LIN {X 0,Y 577.255,Z 419.298,A -85,B 0,C 180,E1 20726.656,E2 20726.656} C_VEL
LIN {X 0,Y 577.259,Z 419.322,A -85,B 0,C 180,E1 20723.262,E2 20723.262} C_VEL
LIN {X 0,Y 577.272,Z 419.276,A -85,B 0,C 180,E1 20720.374,E2 20720.374} C_VEL
LIN {X 0,Y 577.266,Z 419.321,A -85,B 0,C 180,E1 20717.021,E2 20717.021} C_VEL
LIN {X 0,Y 577.313,Z 419.275,A -85,B 0,C 180,E1 20713.931,E2 20713.931} C_VEL
LIN {X 0,Y 577.267,Z 419.299,A -85,B 0,C 180,E1 20710.681,E2 20710.681} C_VEL
LIN {X 0,Y 577.322,Z 419.289,A -85,B 0,C 180,E1 20707.464,E2 20707.464} C_VEL
LIN {X 0,Y 577.275,Z 419.285,A -85,B 0,C 180,E1 20704.271,E2 20704.271} C_VEL
LIN {X 0,Y 577.307,Z 419.309,A -85,B 0,C 180,E1 20700.893,E2 20700.893} C_VEL
LIN {X 0,Y 577.308,Z 419.27,A -85,B 0,C 180,E1 20697.618,E2 20697.618} C_VEL
LIN {X 0,Y 577.29,Z 419.318,A -85,B 0,C 180,E1 20694.334,E2 20694.334} C_VEL
LIN {X 0,Y 577.307,Z 419.266,A -85,B 0,C 180,E1 20691.133,E2 20691.133} C_VEL
LIN {X 0,Y 577.298,Z 419.321,A -85,B 0,C 180,E1 20687.903,E2 20687.903} C_VEL
LIN {X 0,Y 577.31,Z 419.27,A -85,B 0,C 180,E1 20684.633,E2 20684.633} C_VEL
LIN {X 0,Y 577.313,Z 419.303,A -85,B 0,C 180,E1 20681.312,E2 20681.312} C_VEL
LIN {X 0,Y 577.312,Z 419.296,A -85,B 0,C 180,E1 20678.031,E2 20678.031} C_VEL
LIN {X 0,Y 577.295,Z 419.275,A -85,B 0,C 180,E1 20674.781,E2 20674.781} C_VEL
LIN {X 0,Y 577.312,Z 419.307,A -85,B 0,C 180,E1 20671.556,E2 20671.556} C_VEL
LIN {X 0,Y 577.315,Z 419.337,A -85,B 0,C 180,E1 20669.536,E2 20669.536} C_VEL
LIN {X 0,Y 578.617,Z 422.754,A -85,B 0,C 180,E1 20669.207,E2 20669.207} C_VEL
LIN {X 0,Y 581.308,Z 425.275,A -85,B 0,C 180,E1 20668.704,E2 20668.704} C_VEL
LIN {X 0,Y 582.264,Z 426.059,A -85,B 0,C 180,E1 20668.53,E2 20668.53} C_VEL
LIN {X 0,Y 584.624,Z 429.805,A -85,B 0,C 180,E1 20668.068,E2 20668.068} C_VEL
LIN {X 0,Y 587.281,Z 432.33,A -85,B 0,C 180,E1 20667.596,E2 20667.596} C_VEL
LIN {X 0,Y 590.354,Z 436.457,A -85,B 0,C 180,E1 20667.036,E2 20667.036} C_VEL
LIN {X 0,Y 592.909,Z 439.484,A -85,B 0,C 180,E1 20666.591,E2 20666.591} C_VEL
LIN {X 0,Y 603.214,Z 452.791,A -85,B 0,C 180,E1 20664.858,E2 20664.858} C_VEL
LIN {X 0,Y 615.76,Z 470.076,A -85,B 0,C 180,E1 20662.897,E2 20662.897} C_VEL
LIN {X 0,Y 629.647,Z 490.433,A -85,B 0,C 180,E1 20660.888,E2 20660.888} C_VEL
LIN {X 0,Y 623.894,Z 691.807,A -85,B 0,C 180,E1 20658.019,E2 20658.019} C_VEL
LIN {X 0,Y 623.038,Z 722.937,A -85,B 0,C 180,E1 20657.582,E2 20657.582} C_VEL
LIN {X 0,Y 622.123,Z 730.643,A -85,B 0,C 180,E1 20657.545,E2 20657.545} C_VEL
LIN {X 0,Y 617.355,Z 751.291,A -85,B 0,C 180,E1 20657.682,E2 20657.682} C_VEL
LIN {X 0,Y 616.661,Z 757.897,A -85,B 0,C 180,E1 20657.641,E2 20657.641} C_VEL
LIN {X 0,Y 612.677,Z 894.526,A -85,B 0,C 180,E1 20655.715,E2 20655.715} C_VEL
LIN {X 0,Y 611.264,Z 919.339,A -85,B 0,C 180,E1 20655.259,E2 20655.259} C_VEL
LIN {X 0,Y 609.02,Z 947.274,A -85,B 0,C 180,E1 20654.559,E2 20654.559} C_VEL
LIN {X 0,Y 606.96,Z 968.773,A -85,B 0,C 180,E1 20653.88,E2 20653.88} C_VEL
LIN {X 0,Y 604.761,Z 988.806,A -85,B 0,C 180,E1 20653.132,E2 20653.132} C_VEL
LIN {X 0,Y 602.479,Z 1008.004,A -85,B 0,C 180,E1 20652.299,E2 20652.299} C_VEL
LIN {X 0,Y 599.973,Z 1027.016,A -85,B 0,C 180,E1 20651.361,E2 20651.361} C_VEL
LIN {X 0,Y 597.085,Z 1047.482,A -85,B 0,C 180,E1 20650.215,E2 20650.215} C_VEL
LIN {X 0,Y 593.295,Z 1072.796,A -85,B 0,C 180,E1 20648.578,E2 20648.578} C_VEL
LIN {X 0,Y 590.157,Z 1092.691,A -85,B 0,C 180,E1 20647.098,E2 20647.098} C_VEL
LIN {X 0,Y 587.384,Z 1109.948,A -85,B 0,C 180,E1 20645.665,E2 20645.665} C_VEL
LIN {X 0,Y 584.673,Z 1126.712,A -85,B 0,C 180,E1 20644.122,E2 20644.122} C_VEL
LIN {X 0,Y 581.533,Z 1146.472,A -85,B 0,C 180,E1 20642.095,E2 20642.095} C_VEL
LIN {X 0,Y 578.659,Z 1164.633,A -85,B 0,C 180,E1 20639.96,E2 20639.96} C_VEL
LIN {X 0,Y 576.427,Z 1179.555,A -85,B 0,C 180,E1 20638.002,E2 20638.002} C_VEL
LIN {X 0,Y 574.396,Z 1193.881,A -85,B 0,C 180,E1 20635.91,E2 20635.91} C_VEL
LIN {X 0,Y 572.334,Z 1210.036,A -85,B 0,C 180,E1 20633.227,E2 20633.227} C_VEL
LIN {X 0,Y 570.945,Z 1222.042,A -85,B 0,C 180,E1 20630.934,E2 20630.934} C_VEL
LIN {X 0,Y 569.91,Z 1232.241,A -85,B 0,C 180,E1 20628.73,E2 20628.73} C_VEL
LIN {X 0,Y 569.079,Z 1242.76,A -85,B 0,C 180,E1 20626.12,E2 20626.12} C_VEL
LIN {X 0,Y 568.482,Z 1251.696,A -85,B 0,C 180,E1 20623.427,E2 20623.427} C_VEL
LIN {X 0,Y 568.187,Z 1257.937,A -85,B 0,C 180,E1 20621.164,E2 20621.164} C_VEL
LIN {X 0,Y 568.01,Z 1263.03,A -85,B 0,C 180,E1 20618.914,E2 20618.914} C_VEL
LIN {X 0,Y 567.949,Z 1267.415,A -85,B 0,C 180,E1 20616.371,E2 20616.371} C_VEL
LIN {X 0,Y 567.913,Z 1270.438,A -85,B 0,C 180,E1 20613.637,E2 20613.637} C_VEL
LIN {X 0,Y 567.901,Z 1271.703,A -85,B 0,C 180,E1 20611.314,E2 20611.314} C_VEL
LIN {X 0,Y 567.864,Z 1271.838,A -85,B 0,C 180,E1 20609.196,E2 20609.196} C_VEL
LIN {X 0,Y 567.911,Z 1270.98,A -85,B 0,C 180,E1 20607.076,E2 20607.076} C_VEL
LIN {X 0,Y 567.922,Z 1269.047,A -85,B 0,C 180,E1 20604.852,E2 20604.852} C_VEL
LIN {X 0,Y 567.957,Z 1265.815,A -85,B 0,C 180,E1 20602.518,E2 20602.518} C_VEL
LIN {X 0,Y 568.093,Z 1260.701,A -85,B 0,C 180,E1 20599.866,E2 20599.866} C_VEL
LIN {X 0,Y 568.382,Z 1253.797,A -85,B 0,C 180,E1 20597.197,E2 20597.197} C_VEL
LIN {X 0,Y 568.805,Z 1246.674,A -85,B 0,C 180,E1 20594.924,E2 20594.924} C_VEL
LIN {X 0,Y 569.368,Z 1238.677,A -85,B 0,C 180,E1 20592.739,E2 20592.739} C_VEL
LIN {X 0,Y 570.319,Z 1228.371,A -85,B 0,C 180,E1 20590.302,E2 20590.302} C_VEL
LIN {X 0,Y 571.731,Z 1214.972,A -85,B 0,C 180,E1 20587.593,E2 20587.593} C_VEL
LIN {X 0,Y 573.255,Z 1202.375,A -85,B 0,C 180,E1 20585.367,E2 20585.367} C_VEL
LIN {X 0,Y 575.105,Z 1188.883,A -85,B 0,C 180,E1 20583.242,E2 20583.242} C_VEL
LIN {X 0,Y 577.784,Z 1170.42,A -85,B 0,C 180,E1 20580.681,E2 20580.681} C_VEL
LIN {X 0,Y 580.26,Z 1154.409,A -85,B 0,C 180,E1 20578.727,E2 20578.727} C_VEL
LIN {X 0,Y 582.66,Z 1139.203,A -85,B 0,C 180,E1 20577.049,E2 20577.049} C_VEL
LIN {X 0,Y 585.444,Z 1122.069,A -85,B 0,C 180,E1 20575.343,E2 20575.343} C_VEL
LIN {X 0,Y 589.014,Z 1099.841,A -85,B 0,C 180,E1 20573.378,E2 20573.378} C_VEL
LIN {X 0,Y 592.274,Z 1079.106,A -85,B 0,C 180,E1 20571.782,E2 20571.782} C_VEL
LIN {X 0,Y 595.098,Z 1060.635,A -85,B 0,C 180,E1 20570.515,E2 20570.515} C_VEL
LIN {X 0,Y 598.159,Z 1039.88,A -85,B 0,C 180,E1 20569.249,E2 20569.249} C_VEL
LIN {X 0,Y 601.84,Z 1013.091,A -85,B 0,C 180,E1 20567.846,E2 20567.846} C_VEL
LIN {X 0,Y 604.399,Z 992.012,A -85,B 0,C 180,E1 20566.908,E2 20566.908} C_VEL
LIN {X 0,Y 606.726,Z 970.971,A -85,B 0,C 180,E1 20566.107,E2 20566.107} C_VEL
LIN {X 0,Y 608.75,Z 950.092,A -85,B 0,C 180,E1 20565.433,E2 20565.433} C_VEL
LIN {X 0,Y 610.629,Z 927.736,A -85,B 0,C 180,E1 20564.843,E2 20564.843} C_VEL
LIN {X 0,Y 612.456,Z 899.611,A -85,B 0,C 180,E1 20564.274,E2 20564.274} C_VEL
LIN {X 0,Y 614.038,Z 851.534,A -85,B 0,C 180,E1 20563.579,E2 20563.579} C_VEL
LIN {X 0,Y 620.348,Z 631.132,A -85,B 0,C 180,E1 20560.474,E2 20560.474} C_VEL
LIN {X 0,Y 624.432,Z 494.419,A -85,B 0,C 180,E1 20558.499,E2 20558.499} C_VEL
LIN {X 0,Y 611.394,Z 475.211,A -85,B 0,C 180,E1 20556.563,E2 20556.563} C_VEL
LIN {X 0,Y 598.761,Z 457.785,A -85,B 0,C 180,E1 20554.537,E2 20554.537} C_VEL
LIN {X 0,Y 588.143,Z 444.02,A -85,B 0,C 180,E1 20552.697,E2 20552.697} C_VEL
LIN {X 0,Y 584.586,Z 439.654,A -85,B 0,C 180,E1 20552.05,E2 20552.05} C_VEL
LIN {X 0,Y 583.05,Z 437.933,A -85,B 0,C 180,E1 20551.768,E2 20551.768} C_VEL
LIN {X 0,Y 579.933,Z 434.1,A -85,B 0,C 180,E1 20551.177,E2 20551.177} C_VEL
LIN {X 0,Y 578.924,Z 432.665,A -85,B 0,C 180,E1 20550.977,E2 20550.977} C_VEL
LIN {X 0,Y 575.807,Z 429.629,A -85,B 0,C 180,E1 20550.382,E2 20550.382} C_VEL
LIN {X 0,Y 573.999,Z 426.555,A -85,B 0,C 180,E1 20549.997,E2 20549.997} C_VEL
LIN {X 0,Y 571.024,Z 424.302,A -85,B 0,C 180,E1 20549.418,E2 20549.418} C_VEL
LIN {X 0,Y 569.558,Z 421.482,A -85,B 0,C 180,E1 20549.083,E2 20549.083} C_VEL
LIN {X 0,Y 569.316,Z 420.278,A -85,B 0,C 180,E1 20548.996,E2 20548.996} C_VEL
LIN {X 0,Y 569.359,Z 420.26,A -85,B 0,C 180,E1 20545.819,E2 20545.819} C_VEL
LIN {X 0,Y 569.316,Z 420.316,A -85,B 0,C 180,E1 20542.73,E2 20542.73} C_VEL
LIN {X 0,Y 569.344,Z 420.268,A -85,B 0,C 180,E1 20539.44,E2 20539.44} C_VEL
LIN {X 0,Y 569.315,Z 420.29,A -85,B 0,C 180,E1 20536.425,E2 20536.425} C_VEL
LIN {X 0,Y 569.329,Z 420.286,A -85,B 0,C 180,E1 20533.095,E2 20533.095} C_VEL
LIN {X 0,Y 569.315,Z 420.275,A -85,B 0,C 180,E1 20530.115,E2 20530.115} C_VEL
LIN {X 0,Y 569.318,Z 420.302,A -85,B 0,C 180,E1 20526.758,E2 20526.758} C_VEL
LIN {X 0,Y 569.317,Z 420.269,A -85,B 0,C 180,E1 20523.827,E2 20523.827} C_VEL
LIN {X 0,Y 569.314,Z 420.308,A -85,B 0,C 180,E1 20520.503,E2 20520.503} C_VEL
LIN {X 0,Y 569.316,Z 420.267,A -85,B 0,C 180,E1 20517.584,E2 20517.584} C_VEL
LIN {X 0,Y 569.312,Z 420.313,A -85,B 0,C 180,E1 20514.254,E2 20514.254} C_VEL
LIN {X 0,Y 569.312,Z 420.266,A -85,B 0,C 180,E1 20511.38,E2 20511.38} C_VEL
LIN {X 0,Y 569.306,Z 420.314,A -85,B 0,C 180,E1 20508.008,E2 20508.008} C_VEL
LIN {X 0,Y 569.31,Z 420.262,A -85,B 0,C 180,E1 20505.142,E2 20505.142} C_VEL
LIN {X 0,Y 569.303,Z 420.311,A -85,B 0,C 180,E1 20501.782,E2 20501.782} C_VEL
LIN {X 0,Y 569.319,Z 420.264,A -85,B 0,C 180,E1 20498.789,E2 20498.789} C_VEL
LIN {X 0,Y 569.295,Z 420.28,A -85,B 0,C 180,E1 20495.512,E2 20495.512} C_VEL
LIN {X 0,Y 569.333,Z 420.306,A -85,B 0,C 180,E1 20492.475,E2 20492.475} C_VEL
LIN {X 0,Y 569.34,Z 420.481,A -85,B 0,C 180,E1 20491.662,E2 20491.662} C_VEL
LIN {X 0,Y 570.676,Z 423.891,A -85,B 0,C 180,E1 20490.965,E2 20490.965} C_VEL
LIN {X 0,Y 572.177,Z 425.93,A -85,B 0,C 180,E1 20490.446,E2 20490.446} C_VEL
LIN {X 0,Y 575.339,Z 430.215,A -85,B 0,C 180,E1 20489.793,E2 20489.793} C_VEL
LIN {X 0,Y 577.584,Z 432.958,A -85,B 0,C 180,E1 20489.348,E2 20489.348} C_VEL
LIN {X 0,Y 585.42,Z 442.842,A -85,B 0,C 180,E1 20487.857,E2 20487.857} C_VEL
LIN {X 0,Y 590.299,Z 449.247,A -85,B 0,C 180,E1 20486.972,E2 20486.972} C_VEL
LIN {X 0,Y 600.49,Z 462.84,A -85,B 0,C 180,E1 20485.228,E2 20485.228} C_VEL
LIN {X 0,Y 612.268,Z 479.558,A -85,B 0,C 180,E1 20483.352,E2 20483.352} C_VEL
LIN {X 0,Y 624.192,Z 497.277,A -85,B 0,C 180,E1 20481.586,E2 20481.586} C_VEL
LIN {X 0,Y 624.554,Z 498.373,A -85,B 0,C 180,E1 20481.524,E2 20481.524} C_VEL
LIN {X 0,Y 618.433,Z 702.963,A -85,B 0,C 180,E1 20478.594,E2 20478.594} C_VEL
LIN {X 0,Y 612.66,Z 903.345,A -85,B 0,C 180,E1 20475.772,E2 20475.772} C_VEL
LIN {X 0,Y 611.318,Z 926.912,A -85,B 0,C 180,E1 20475.346,E2 20475.346} C_VEL
LIN {X 0,Y 609.063,Z 955.797,A -85,B 0,C 180,E1 20474.637,E2 20474.637} C_VEL
LIN {X 0,Y 606.994,Z 977.545,A -85,B 0,C 180,E1 20473.957,E2 20473.957} C_VEL
LIN {X 0,Y 604.718,Z 998.44,A -85,B 0,C 180,E1 20473.182,E2 20473.182} C_VEL
LIN {X 0,Y 602.468,Z 1017.534,A -85,B 0,C 180,E1 20472.356,E2 20472.356} C_VEL
LIN {X 0,Y 599.952,Z 1036.808,A -85,B 0,C 180,E1 20471.411,E2 20471.411} C_VEL
LIN {X 0,Y 597.09,Z 1057.377,A -85,B 0,C 180,E1 20470.265,E2 20470.265} C_VEL
LIN {X 0,Y 593.319,Z 1082.691,A -85,B 0,C 180,E1 20468.631,E2 20468.631} C_VEL
LIN {X 0,Y 590.173,Z 1102.602,A -85,B 0,C 180,E1 20467.151,E2 20467.151} C_VEL
LIN {X 0,Y 587.38,Z 1119.973,A -85,B 0,C 180,E1 20465.709,E2 20465.709} C_VEL
LIN {X 0,Y 584.596,Z 1137.198,A -85,B 0,C 180,E1 20464.12,E2 20464.12} C_VEL
LIN {X 0,Y 581.466,Z 1156.906,A -85,B 0,C 180,E1 20462.092,E2 20462.092} C_VEL
LIN {X 0,Y 578.6,Z 1175.014,A -85,B 0,C 180,E1 20459.957,E2 20459.957} C_VEL
LIN {X 0,Y 576.36,Z 1189.974,A -85,B 0,C 180,E1 20457.989,E2 20457.989} C_VEL
LIN {X 0,Y 574.263,Z 1204.905,A -85,B 0,C 180,E1 20455.799,E2 20455.799} C_VEL
LIN {X 0,Y 572.246,Z 1220.722,A -85,B 0,C 180,E1 20453.146,E2 20453.146} C_VEL
LIN {X 0,Y 570.918,Z 1232.282,A -85,B 0,C 180,E1 20450.929,E2 20450.929} C_VEL
LIN {X 0,Y 569.931,Z 1242,A -85,B 0,C 180,E1 20448.829,E2 20448.829} C_VEL
LIN {X 0,Y 569.148,Z 1251.779,A -85,B 0,C 180,E1 20446.417,E2 20446.417} C_VEL
LIN {X 0,Y 568.498,Z 1261.236,A -85,B 0,C 180,E1 20443.628,E2 20443.628} C_VEL
LIN {X 0,Y 568.204,Z 1267.555,A -85,B 0,C 180,E1 20441.363,E2 20441.363} C_VEL
LIN {X 0,Y 568.006,Z 1272.72,A -85,B 0,C 180,E1 20439.112,E2 20439.112} C_VEL
LIN {X 0,Y 567.949,Z 1276.862,A -85,B 0,C 180,E1 20436.771,E2 20436.771} C_VEL
LIN {X 0,Y 567.919,Z 1280.098,A -85,B 0,C 180,E1 20434.136,E2 20434.136} C_VEL
LIN {X 0,Y 567.902,Z 1281.691,A -85,B 0,C 180,E1 20431.409,E2 20431.409} C_VEL
LIN {X 0,Y 567.864,Z 1281.849,A -85,B 0,C 180,E1 20429.291,E2 20429.291} C_VEL
LIN {X 0,Y 567.911,Z 1281.013,A -85,B 0,C 180,E1 20427.172,E2 20427.172} C_VEL
LIN {X 0,Y 567.921,Z 1279.102,A -85,B 0,C 180,E1 20424.947,E2 20424.947} C_VEL
LIN {X 0,Y 567.957,Z 1275.894,A -85,B 0,C 180,E1 20422.614,E2 20422.614} C_VEL
LIN {X 0,Y 568.085,Z 1270.812,A -85,B 0,C 180,E1 20419.962,E2 20419.962} C_VEL
LIN {X 0,Y 568.369,Z 1263.95,A -85,B 0,C 180,E1 20417.294,E2 20417.294} C_VEL
LIN {X 0,Y 568.792,Z 1256.852,A -85,B 0,C 180,E1 20415.022,E2 20415.022} C_VEL
LIN {X 0,Y 569.352,Z 1248.81,A -85,B 0,C 180,E1 20412.818,E2 20412.818} C_VEL
LIN {X 0,Y 570.279,Z 1238.756,A -85,B 0,C 180,E1 20410.432,E2 20410.432} C_VEL
LIN {X 0,Y 571.697,Z 1225.279,A -85,B 0,C 180,E1 20407.693,E2 20407.693} C_VEL
LIN {X 0,Y 573.209,Z 1212.716,A -85,B 0,C 180,E1 20405.469,E2 20405.469} C_VEL
LIN {X 0,Y 575.051,Z 1199.261,A -85,B 0,C 180,E1 20403.344,E2 20403.344} C_VEL
LIN {X 0,Y 577.59,Z 1181.727,A -85,B 0,C 180,E1 20400.891,E2 20400.891} C_VEL
LIN {X 0,Y 580.209,Z 1164.739,A -85,B 0,C 180,E1 20398.81,E2 20398.81} C_VEL
LIN {X 0,Y 582.65,Z 1149.263,A -85,B 0,C 180,E1 20397.1,E2 20397.1} C_VEL
LIN {X 0,Y 585.394,Z 1132.354,A -85,B 0,C 180,E1 20395.416,E2 20395.416} C_VEL
LIN {X 0,Y 588.911,Z 1110.53,A -85,B 0,C 180,E1 20393.479,E2 20393.479} C_VEL
LIN {X 0,Y 592.253,Z 1089.208,A -85,B 0,C 180,E1 20391.835,E2 20391.835} C_VEL
LIN {X 0,Y 595.075,Z 1070.76,A -85,B 0,C 180,E1 20390.568,E2 20390.568} C_VEL
LIN {X 0,Y 597.874,Z 1051.659,A -85,B 0,C 180,E1 20389.401,E2 20389.401} C_VEL
LIN {X 0,Y 601.073,Z 1028.507,A -85,B 0,C 180,E1 20388.158,E2 20388.158} C_VEL
LIN {X 0,Y 604.185,Z 1003.202,A -85,B 0,C 180,E1 20387.011,E2 20387.011} C_VEL
LIN {X 0,Y 606.568,Z 981.579,A -85,B 0,C 180,E1 20386.183,E2 20386.183} C_VEL
LIN {X 0,Y 608.634,Z 960.325,A -85,B 0,C 180,E1 20385.495,E2 20385.495} C_VEL
LIN {X 0,Y 610.45,Z 938.806,A -85,B 0,C 180,E1 20384.923,E2 20384.923} C_VEL
LIN {X 0,Y 612.158,Z 913.923,A -85,B 0,C 180,E1 20384.401,E2 20384.401} C_VEL
LIN {X 0,Y 613.575,Z 876.43,A -85,B 0,C 180,E1 20383.838,E2 20383.838} C_VEL
LIN {X 0,Y 619.924,Z 652.053,A -85,B 0,C 180,E1 20380.685,E2 20380.685} C_VEL
LIN {X 0,Y 624.525,Z 497.803,A -85,B 0,C 180,E1 20378.463,E2 20378.463} C_VEL
LIN {X 0,Y 612.514,Z 479.937,A -85,B 0,C 180,E1 20376.689,E2 20376.689} C_VEL
LIN {X 0,Y 601.717,Z 464.605,A -85,B 0,C 180,E1 20374.981,E2 20374.981} C_VEL
LIN {X 0,Y 595.232,Z 455.876,A -85,B 0,C 180,E1 20373.897,E2 20373.897} C_VEL
LIN {X 0,Y 587.981,Z 446.173,A -85,B 0,C 180,E1 20372.621,E2 20372.621} C_VEL
LIN {X 0,Y 579.919,Z 435.911,A -85,B 0,C 180,E1 20371.12,E2 20371.12} C_VEL
LIN {X 0,Y 575.515,Z 430.361,A -85,B 0,C 180,E1 20370.255,E2 20370.255} C_VEL
LIN {X 0,Y 572.223,Z 426.049,A -85,B 0,C 180,E1 20369.58,E2 20369.58} C_VEL
LIN {X 0,Y 571.22,Z 424.558,A -85,B 0,C 180,E1 20369.234,E2 20369.234} C_VEL
LIN {X 0,Y 569.558,Z 421.437,A -85,B 0,C 180,E1 20368.523,E2 20368.523} C_VEL
LIN {X 0,Y 569.355,Z 420.292,A -85,B 0,C 180,E1 20368.305,E2 20368.305} C_VEL
LIN {X 0,Y 569.307,Z 420.267,A -85,B 0,C 180,E1 20365.153,E2 20365.153} C_VEL
LIN {X 0,Y 569.386,Z 420.287,A -85,B 0,C 180,E1 20361.965,E2 20361.965} C_VEL
LIN {X 0,Y 569.317,Z 420.29,A -85,B 0,C 180,E1 20358.748,E2 20358.748} C_VEL
LIN {X 0,Y 569.378,Z 420.258,A -85,B 0,C 180,E1 20355.586,E2 20355.586} C_VEL
LIN {X 0,Y 569.335,Z 420.309,A -85,B 0,C 180,E1 20352.372,E2 20352.372} C_VEL
LIN {X 0,Y 569.342,Z 420.255,A -85,B 0,C 180,E1 20348.992,E2 20348.992} C_VEL
LIN {X 0,Y 569.37,Z 420.309,A -85,B 0,C 180,E1 20345.846,E2 20345.846} C_VEL
LIN {X 0,Y 569.336,Z 420.258,A -85,B 0,C 180,E1 20342.516,E2 20342.516} C_VEL
LIN {X 0,Y 569.38,Z 420.299,A -85,B 0,C 180,E1 20339.296,E2 20339.296} C_VEL
LIN {X 0,Y 569.35,Z 420.263,A -85,B 0,C 180,E1 20335.964,E2 20335.964} C_VEL
LIN {X 0,Y 569.372,Z 420.285,A -85,B 0,C 180,E1 20332.635,E2 20332.635} C_VEL
LIN {X 0,Y 569.372,Z 420.279,A -85,B 0,C 180,E1 20329.272,E2 20329.272} C_VEL
LIN {X 0,Y 569.356,Z 420.267,A -85,B 0,C 180,E1 20325.974,E2 20325.974} C_VEL
LIN {X 0,Y 569.37,Z 420.305,A -85,B 0,C 180,E1 20322.735,E2 20322.735} C_VEL
LIN {X 0,Y 569.373,Z 420.258,A -85,B 0,C 180,E1 20319.33,E2 20319.33} C_VEL
LIN {X 0,Y 569.375,Z 420.286,A -85,B 0,C 180,E1 20316.067,E2 20316.067} C_VEL
LIN {X 0,Y 569.36,Z 420.294,A -85,B 0,C 180,E1 20312.701,E2 20312.701} C_VEL
LIN {X 0,Y 569.379,Z 420.415,A -85,B 0,C 180,E1 20310.87,E2 20310.87} C_VEL
LIN {X 0,Y 570.427,Z 423.392,A -85,B 0,C 180,E1 20310.606,E2 20310.606} C_VEL
LIN {X 0,Y 572.868,Z 425.927,A -85,B 0,C 180,E1 20310.111,E2 20310.111} C_VEL
LIN {X 0,Y 574.435,Z 427.024,A -85,B 0,C 180,E1 20309.812,E2 20309.812} C_VEL
LIN {X 0,Y 576.752,Z 430.772,A -85,B 0,C 180,E1 20309.327,E2 20309.327} C_VEL
LIN {X 0,Y 579.551,Z 433.39,A -85,B 0,C 180,E1 20308.801,E2 20308.801} C_VEL
LIN {X 0,Y 582.512,Z 437.438,A -85,B 0,C 180,E1 20308.228,E2 20308.228} C_VEL
LIN {X 0,Y 584.579,Z 439.588,A -85,B 0,C 180,E1 20307.852,E2 20307.852} C_VEL
LIN {X 0,Y 588.094,Z 443.946,A -85,B 0,C 180,E1 20307.213,E2 20307.213} C_VEL
LIN {X 0,Y 597.347,Z 455.975,A -85,B 0,C 180,E1 20305.602,E2 20305.602} C_VEL
LIN {X 0,Y 609.156,Z 472.052,A -85,B 0,C 180,E1 20303.69,E2 20303.69} C_VEL
LIN {X 0,Y 620.362,Z 488.375,A -85,B 0,C 180,E1 20301.997,E2 20301.997} C_VEL
LIN {X 0,Y 624.49,Z 494.843,A -85,B 0,C 180,E1 20301.396,E2 20301.396} C_VEL
LIN {X 0,Y 618.135,Z 706.554,A -85,B 0,C 180,E1 20298.365,E2 20298.365} C_VEL
LIN {X 0,Y 616.661,Z 757.897,A -85,B 0,C 180,E1 20297.641,E2 20297.641} C_VEL
LIN {X 0,Y 615.763,Z 765.6,A -85,B 0,C 180,E1 20297.602,E2 20297.602} C_VEL
LIN {X 0,Y 610.953,Z 786.238,A -85,B 0,C 180,E1 20297.745,E2 20297.745} C_VEL
LIN {X 0,Y 610.243,Z 792.846,A -85,B 0,C 180,E1 20297.705,E2 20297.705} C_VEL
LIN {X 0,Y 607.082,Z 895.175,A -85,B 0,C 180,E1 20296.248,E2 20296.248} C_VEL
LIN {X 0,Y 605.476,Z 922.029,A -85,B 0,C 180,E1 20295.747,E2 20295.747} C_VEL
LIN {X 0,Y 603.194,Z 948.425,A -85,B 0,C 180,E1 20295.066,E2 20295.066} C_VEL
LIN {X 0,Y 601.07,Z 969.618,A -85,B 0,C 180,E1 20294.389,E2 20294.389} C_VEL
LIN {X 0,Y 598.702,Z 990.192,A -85,B 0,C 180,E1 20293.611,E2 20293.611} C_VEL
LIN {X 0,Y 596.112,Z 1010.852,A -85,B 0,C 180,E1 20292.698,E2 20292.698} C_VEL
LIN {X 0,Y 592.764,Z 1035.101,A -85,B 0,C 180,E1 20291.46,E2 20291.46} C_VEL
LIN {X 0,Y 589.089,Z 1058.632,A -85,B 0,C 180,E1 20290.039,E2 20290.039} C_VEL
LIN {X 0,Y 586.085,Z 1077.213,A -85,B 0,C 180,E1 20288.766,E2 20288.766} C_VEL
LIN {X 0,Y 583.082,Z 1095.367,A -85,B 0,C 180,E1 20287.378,E2 20287.378} C_VEL
LIN {X 0,Y 579.896,Z 1114.212,A -85,B 0,C 180,E1 20285.771,E2 20285.771} C_VEL
LIN {X 0,Y 576.121,Z 1136.346,A -85,B 0,C 180,E1 20283.619,E2 20283.619} C_VEL
LIN {X 0,Y 573.324,Z 1152.994,A -85,B 0,C 180,E1 20281.784,E2 20281.784} C_VEL
LIN {X 0,Y 570.852,Z 1168.016,A -85,B 0,C 180,E1 20279.949,E2 20279.949} C_VEL
LIN {X 0,Y 568.127,Z 1185.441,A -85,B 0,C 180,E1 20277.575,E2 20277.575} C_VEL
LIN {X 0,Y 565.828,Z 1201.189,A -85,B 0,C 180,E1 20275.096,E2 20275.096} C_VEL
LIN {X 0,Y 564.233,Z 1213.323,A -85,B 0,C 180,E1 20272.948,E2 20272.948} C_VEL
LIN {X 0,Y 562.838,Z 1225.244,A -85,B 0,C 180,E1 20270.573,E2 20270.573} C_VEL
LIN {X 0,Y 561.603,Z 1237.509,A -85,B 0,C 180,E1 20267.725,E2 20267.725} C_VEL
LIN {X 0,Y 560.906,Z 1246.241,A -85,B 0,C 180,E1 20265.332,E2 20265.332} C_VEL
LIN {X 0,Y 560.455,Z 1253.303,A -85,B 0,C 180,E1 20263.067,E2 20263.067} C_VEL
LIN {X 0,Y 560.157,Z 1259.718,A -85,B 0,C 180,E1 20260.597,E2 20260.597} C_VEL
LIN {X 0,Y 559.957,Z 1265.342,A -85,B 0,C 180,E1 20257.802,E2 20257.802} C_VEL
LIN {X 0,Y 559.926,Z 1268.822,A -85,B 0,C 180,E1 20255.331,E2 20255.331} C_VEL
LIN {X 0,Y 559.91,Z 1270.847,A -85,B 0,C 180,E1 20253.074,E2 20253.074} C_VEL
LIN {X 0,Y 559.881,Z 1271.771,A -85,B 0,C 180,E1 20251.026,E2 20251.026} C_VEL
LIN {X 0,Y 559.873,Z 1271.792,A -85,B 0,C 180,E1 20248.98,E2 20248.98} C_VEL
LIN {X 0,Y 559.911,Z 1270.911,A -85,B 0,C 180,E1 20246.932,E2 20246.932} C_VEL
LIN {X 0,Y 559.923,Z 1268.929,A -85,B 0,C 180,E1 20244.675,E2 20244.675} C_VEL
LIN {X 0,Y 559.96,Z 1265.491,A -85,B 0,C 180,E1 20242.204,E2 20242.204} C_VEL
LIN {X 0,Y 560.149,Z 1259.953,A -85,B 0,C 180,E1 20239.409,E2 20239.409} C_VEL
LIN {X 0,Y 560.448,Z 1253.492,A -85,B 0,C 180,E1 20236.908,E2 20236.908} C_VEL
LIN {X 0,Y 560.896,Z 1246.318,A -85,B 0,C 180,E1 20234.6,E2 20234.6} C_VEL
LIN {X 0,Y 561.573,Z 1237.862,A -85,B 0,C 180,E1 20232.278,E2 20232.278} C_VEL
LIN {X 0,Y 562.803,Z 1225.581,A -85,B 0,C 180,E1 20229.408,E2 20229.408} C_VEL
LIN {X 0,Y 564.168,Z 1213.82,A -85,B 0,C 180,E1 20227.055,E2 20227.055} C_VEL
LIN {X 0,Y 565.745,Z 1201.734,A -85,B 0,C 180,E1 20224.906,E2 20224.906} C_VEL
LIN {X 0,Y 567.92,Z 1186.761,A -85,B 0,C 180,E1 20222.535,E2 20222.535} C_VEL
LIN {X 0,Y 570.616,Z 1169.546,A -85,B 0,C 180,E1 20220.157,E2 20220.157} C_VEL
LIN {X 0,Y 573.088,Z 1154.433,A -85,B 0,C 180,E1 20218.294,E2 20218.294} C_VEL
LIN {X 0,Y 575.716,Z 1138.688,A -85,B 0,C 180,E1 20216.54,E2 20216.54} C_VEL
LIN {X 0,Y 578.848,Z 1120.395,A -85,B 0,C 180,E1 20214.709,E2 20214.709} C_VEL
LIN {X 0,Y 582.679,Z 1097.76,A -85,B 0,C 180,E1 20212.722,E2 20212.722} C_VEL
LIN {X 0,Y 585.811,Z 1078.871,A -85,B 0,C 180,E1 20211.264,E2 20211.264} C_VEL
LIN {X 0,Y 588.794,Z 1060.419,A -85,B 0,C 180,E1 20209.986,E2 20209.986} C_VEL
LIN {X 0,Y 591.945,Z 1040.055,A -85,B 0,C 180,E1 20208.736,E2 20208.736} C_VEL
LIN {X 0,Y 595.666,Z 1014.294,A -85,B 0,C 180,E1 20207.372,E2 20207.372} C_VEL
LIN {X 0,Y 598.557,Z 991.428,A -85,B 0,C 180,E1 20206.349,E2 20206.349} C_VEL
LIN {X 0,Y 600.915,Z 971.041,A -85,B 0,C 180,E1 20205.571,E2 20205.571} C_VEL
LIN {X 0,Y 603.032,Z 950.05,A -85,B 0,C 180,E1 20204.891,E2 20204.891} C_VEL
LIN {X 0,Y 604.996,Z 927.537,A -85,B 0,C 180,E1 20204.295,E2 20204.295} C_VEL
LIN {X 0,Y 606.923,Z 898.692,A -85,B 0,C 180,E1 20203.716,E2 20203.716} C_VEL
LIN {X 0,Y 608.642,Z 847.708,A -85,B 0,C 180,E1 20202.977,E2 20202.977} C_VEL
LIN {X 0,Y 615.268,Z 627.748,A -85,B 0,C 180,E1 20199.856,E2 20199.856} C_VEL
LIN {X 0,Y 619.331,Z 498.457,A -85,B 0,C 180,E1 20197.975,E2 20197.975} C_VEL
LIN {X 0,Y 606.402,Z 479.36,A -85,B 0,C 180,E1 20196.003,E2 20196.003} C_VEL
LIN {X 0,Y 592.009,Z 459.543,A -85,B 0,C 180,E1 20193.612,E2 20193.612} C_VEL
LIN {X 0,Y 585.035,Z 450.699,A -85,B 0,C 180,E1 20192.37,E2 20192.37} C_VEL
LIN {X 0,Y 580.351,Z 444.972,A -85,B 0,C 180,E1 20191.498,E2 20191.498} C_VEL
LIN {X 0,Y 576.818,Z 440.49,A -85,B 0,C 180,E1 20190.813,E2 20190.813} C_VEL
LIN {X 0,Y 572.742,Z 436.034,A -85,B 0,C 180,E1 20190.011,E2 20190.011} C_VEL
LIN {X 0,Y 571.245,Z 433.754,A -85,B 0,C 180,E1 20189.693,E2 20189.693} C_VEL
LIN {X 0,Y 568.122,Z 430.903,A -85,B 0,C 180,E1 20189.062,E2 20189.062} C_VEL
LIN {X 0,Y 566.3,Z 427.687,A -85,B 0,C 180,E1 20188.645,E2 20188.645} C_VEL
LIN {X 0,Y 563.23,Z 425.419,A -85,B 0,C 180,E1 20188.006,E2 20188.006} C_VEL
LIN {X 0,Y 561.67,Z 422.586,A -85,B 0,C 180,E1 20187.628,E2 20187.628} C_VEL
LIN {X 0,Y 561.392,Z 421.296,A -85,B 0,C 180,E1 20187.515,E2 20187.515} C_VEL
LIN {X 0,Y 561.401,Z 421.258,A -85,B 0,C 180,E1 20184.407,E2 20184.407} C_VEL
LIN {X 0,Y 561.379,Z 421.26,A -85,B 0,C 180,E1 20181.197,E2 20181.197} C_VEL
LIN {X 0,Y 561.406,Z 421.291,A -85,B 0,C 180,E1 20178.161,E2 20178.161} C_VEL
LIN {X 0,Y 561.366,Z 421.247,A -85,B 0,C 180,E1 20174.862,E2 20174.862} C_VEL
LIN {X 0,Y 561.417,Z 421.301,A -85,B 0,C 180,E1 20171.819,E2 20171.819} C_VEL
LIN {X 0,Y 561.363,Z 421.247,A -85,B 0,C 180,E1 20168.605,E2 20168.605} C_VEL
LIN {X 0,Y 561.411,Z 421.3,A -85,B 0,C 180,E1 20165.622,E2 20165.622} C_VEL
LIN {X 0,Y 561.36,Z 421.249,A -85,B 0,C 180,E1 20162.348,E2 20162.348} C_VEL
LIN {X 0,Y 561.423,Z 421.294,A -85,B 0,C 180,E1 20159.286,E2 20159.286} C_VEL
LIN {X 0,Y 561.356,Z 421.253,A -85,B 0,C 180,E1 20156.017,E2 20156.017} C_VEL
LIN {X 0,Y 561.441,Z 421.284,A -85,B 0,C 180,E1 20152.839,E2 20152.839} C_VEL
LIN {X 0,Y 561.354,Z 421.26,A -85,B 0,C 180,E1 20149.636,E2 20149.636} C_VEL
LIN {X 0,Y 561.406,Z 421.269,A -85,B 0,C 180,E1 20146.403,E2 20146.403} C_VEL
LIN {X 0,Y 561.356,Z 421.272,A -85,B 0,C 180,E1 20143.373,E2 20143.373} C_VEL
LIN {X 0,Y 561.392,Z 421.249,A -85,B 0,C 180,E1 20140.112,E2 20140.112} C_VEL
LIN {X 0,Y 561.356,Z 421.303,A -85,B 0,C 180,E1 20137.151,E2 20137.151} C_VEL
LIN {X 0,Y 561.386,Z 421.255,A -85,B 0,C 180,E1 20133.842,E2 20133.842} C_VEL
LIN {X 0,Y 561.362,Z 421.364,A -85,B 0,C 180,E1 20133.059,E2 20133.059} C_VEL
LIN {X 0,Y 562.59,Z 424.593,A -85,B 0,C 180,E1 20132.362,E2 20132.362} C_VEL
LIN {X 0,Y 564.373,Z 426.58,A -85,B 0,C 180,E1 20131.854,E2 20131.854} C_VEL
LIN {X 0,Y 567.267,Z 430.737,A -85,B 0,C 180,E1 20131.207,E2 20131.207} C_VEL
LIN {X 0,Y 569.664,Z 433.205,A -85,B 0,C 180,E1 20130.71,E2 20130.71} C_VEL
LIN {X 0,Y 573.277,Z 437.799,A -85,B 0,C 180,E1 20129.962,E2 20129.962} C_VEL
LIN {X 0,Y 582.806,Z 450.095,A -85,B 0,C 180,E1 20128.101,E2 20128.101} C_VEL
LIN {X 0,Y 587.875,Z 456.785,A -85,B 0,C 180,E1 20127.17,E2 20127.17} C_VEL
LIN {X 0,Y 597.266,Z 469.415,A -85,B 0,C 180,E1 20125.538,E2 20125.538} C_VEL
LIN {X 0,Y 610.901,Z 488.879,A -85,B 0,C 180,E1 20123.344,E2 20123.344} C_VEL
LIN {X 0,Y 619.452,Z 502.2,A -85,B 0,C 180,E1 20122.05,E2 20122.05} C_VEL
LIN {X 0,Y 612.928,Z 710.012,A -85,B 0,C 180,E1 20119.056,E2 20119.056} C_VEL
LIN {X 0,Y 607.076,Z 903.364,A -85,B 0,C 180,E1 20116.313,E2 20116.313} C_VEL
LIN {X 0,Y 605.654,Z 927.281,A -85,B 0,C 180,E1 20115.879,E2 20115.879} C_VEL
LIN {X 0,Y 603.313,Z 955.925,A -85,B 0,C 180,E1 20115.17,E2 20115.17} C_VEL
LIN {X 0,Y 601.092,Z 978.171,A -85,B 0,C 180,E1 20114.469,E2 20114.469} C_VEL
LIN {X 0,Y 598.818,Z 998.119,A -85,B 0,C 180,E1 20113.725,E2 20113.725} C_VEL
LIN {X 0,Y 596.436,Z 1017.445,A -85,B 0,C 180,E1 20112.887,E2 20112.887} C_VEL
LIN {X 0,Y 593.811,Z 1036.588,A -85,B 0,C 180,E1 20111.944,E2 20111.944} C_VEL
LIN {X 0,Y 590.792,Z 1057.286,A -85,B 0,C 180,E1 20110.784,E2 20110.784} C_VEL
LIN {X 0,Y 586.87,Z 1082.596,A -85,B 0,C 180,E1 20109.142,E2 20109.142} C_VEL
LIN {X 0,Y 583.61,Z 1102.282,A -85,B 0,C 180,E1 20107.67,E2 20107.67} C_VEL
LIN {X 0,Y 580.743,Z 1119.26,A -85,B 0,C 180,E1 20106.252,E2 20106.252} C_VEL
LIN {X 0,Y 577.872,Z 1136.087,A -85,B 0,C 180,E1 20104.694,E2 20104.694} C_VEL
LIN {X 0,Y 574.954,Z 1153.291,A -85,B 0,C 180,E1 20102.924,E2 20102.924} C_VEL
LIN {X 0,Y 571.461,Z 1174.167,A -85,B 0,C 180,E1 20100.487,E2 20100.487} C_VEL
LIN {X 0,Y 569.141,Z 1188.863,A -85,B 0,C 180,E1 20098.541,E2 20098.541} C_VEL
LIN {X 0,Y 567.023,Z 1202.801,A -85,B 0,C 180,E1 20096.492,E2 20096.492} C_VEL
LIN {X 0,Y 564.886,Z 1218.401,A -85,B 0,C 180,E1 20093.908,E2 20093.908} C_VEL
LIN {X 0,Y 563.262,Z 1231.25,A -85,B 0,C 180,E1 20091.446,E2 20091.446} C_VEL
LIN {X 0,Y 562.196,Z 1241.081,A -85,B 0,C 180,E1 20089.314,E2 20089.314} C_VEL
LIN {X 0,Y 561.357,Z 1250.123,A -85,B 0,C 180,E1 20087.088,E2 20087.088} C_VEL
LIN {X 0,Y 560.697,Z 1258.993,A -85,B 0,C 180,E1 20084.559,E2 20084.559} C_VEL
LIN {X 0,Y 560.264,Z 1267.044,A -85,B 0,C 180,E1 20081.735,E2 20081.735} C_VEL
LIN {X 0,Y 560.02,Z 1272.304,A -85,B 0,C 180,E1 20079.451,E2 20079.451} C_VEL
LIN {X 0,Y 559.967,Z 1276.38,A -85,B 0,C 180,E1 20077.177,E2 20077.177} C_VEL
LIN {X 0,Y 559.919,Z 1279.448,A -85,B 0,C 180,E1 20074.811,E2 20074.811} C_VEL
LIN {X 0,Y 559.911,Z 1281.55,A -85,B 0,C 180,E1 20072.044,E2 20072.044} C_VEL
LIN {X 0,Y 559.865,Z 1281.871,A -85,B 0,C 180,E1 20069.383,E2 20069.383} C_VEL
LIN {X 0,Y 559.909,Z 1281.081,A -85,B 0,C 180,E1 20067.233,E2 20067.233} C_VEL
LIN {X 0,Y 559.921,Z 1279.213,A -85,B 0,C 180,E1 20064.977,E2 20064.977} C_VEL
LIN {X 0,Y 559.964,Z 1276.21,A -85,B 0,C 180,E1 20062.714,E2 20062.714} C_VEL
LIN {X 0,Y 560.051,Z 1271.672,A -85,B 0,C 180,E1 20060.232,E2 20060.232} C_VEL
LIN {X 0,Y 560.377,Z 1264.556,A -85,B 0,C 180,E1 20057.32,E2 20057.32} C_VEL
LIN {X 0,Y 560.864,Z 1256.852,A -85,B 0,C 180,E1 20054.805,E2 20054.805} C_VEL
LIN {X 0,Y 561.467,Z 1248.885,A -85,B 0,C 180,E1 20052.589,E2 20052.589} C_VEL
LIN {X 0,Y 562.466,Z 1238.758,A -85,B 0,C 180,E1 20050.149,E2 20050.149} C_VEL
LIN {X 0,Y 563.987,Z 1225.278,A -85,B 0,C 180,E1 20047.372,E2 20047.372} C_VEL
LIN {X 0,Y 565.606,Z 1212.714,A -85,B 0,C 180,E1 20045.117,E2 20045.117} C_VEL
LIN {X 0,Y 567.556,Z 1199.259,A -85,B 0,C 180,E1 20042.963,E2 20042.963} C_VEL
LIN {X 0,Y 570.365,Z 1181.123,A -85,B 0,C 180,E1 20040.404,E2 20040.404} C_VEL
LIN {X 0,Y 573.033,Z 1164.761,A -85,B 0,C 180,E1 20038.377,E2 20038.377} C_VEL
LIN {X 0,Y 575.569,Z 1149.569,A -85,B 0,C 180,E1 20036.679,E2 20036.679} C_VEL
LIN {X 0,Y 578.36,Z 1133.256,A -85,B 0,C 180,E1 20035.032,E2 20035.032} C_VEL
LIN {X 0,Y 581.912,Z 1112.493,A -85,B 0,C 180,E1 20033.152,E2 20033.152} C_VEL
LIN {X 0,Y 585.63,Z 1089.94,A -85,B 0,C 180,E1 20031.386,E2 20031.386} C_VEL
LIN {X 0,Y 588.573,Z 1071.512,A -85,B 0,C 180,E1 20030.109,E2 20030.109} C_VEL
LIN {X 0,Y 591.598,Z 1051.765,A -85,B 0,C 180,E1 20028.892,E2 20028.892} C_VEL
LIN {X 0,Y 594.829,Z 1029.426,A -85,B 0,C 180,E1 20027.682,E2 20027.682} C_VEL
LIN {X 0,Y 598.234,Z 1003.121,A -85,B 0,C 180,E1 20026.478,E2 20026.478} C_VEL
LIN {X 0,Y 600.73,Z 981.491,A -85,B 0,C 180,E1 20025.646,E2 20025.646} C_VEL
LIN {X 0,Y 602.862,Z 960.442,A -85,B 0,C 180,E1 20024.962,E2 20024.962} C_VEL
LIN {X 0,Y 604.75,Z 939.042,A -85,B 0,C 180,E1 20024.389,E2 20024.389} C_VEL
LIN {X 0,Y 606.474,Z 914.973,A -85,B 0,C 180,E1 20023.879,E2 20023.879} C_VEL
LIN {X 0,Y 607.97,Z 878.645,A -85,B 0,C 180,E1 20023.324,E2 20023.324} C_VEL
LIN {X 0,Y 614.641,Z 654.12,A -85,B 0,C 180,E1 20020.147,E2 20020.147} C_VEL
LIN {X 0,Y 619.41,Z 501.851,A -85,B 0,C 180,E1 20017.94,E2 20017.94} C_VEL
LIN {X 0,Y 606.991,Z 483.206,A -85,B 0,C 180,E1 20016.05,E2 20016.05} C_VEL
LIN {X 0,Y 593.948,Z 464.767,A -85,B 0,C 180,E1 20013.902,E2 20013.902} C_VEL
LIN {X 0,Y 584.636,Z 452.504,A -85,B 0,C 180,E1 20012.25,E2 20012.25} C_VEL
LIN {X 0,Y 577.014,Z 442.679,A -85,B 0,C 180,E1 20010.802,E2 20010.802} C_VEL
LIN {X 0,Y 572.543,Z 437.042,A -85,B 0,C 180,E1 20009.907,E2 20009.907} C_VEL
LIN {X 0,Y 568.638,Z 431.999,A -85,B 0,C 180,E1 20009.091,E2 20009.091} C_VEL
LIN {X 0,Y 565.309,Z 428.206,A -85,B 0,C 180,E1 20008.382,E2 20008.382} C_VEL
LIN {X 0,Y 563.876,Z 426.106,A -85,B 0,C 180,E1 20008.057,E2 20008.057} C_VEL
LIN {X 0,Y 561.693,Z 422.759,A -85,B 0,C 180,E1 20007.226,E2 20007.226} C_VEL
LIN {X 0,Y 561.367,Z 421.281,A -85,B 0,C 180,E1 20006.899,E2 20006.899} C_VEL
LIN {X 0,Y 561.41,Z 421.279,A -85,B 0,C 180,E1 20003.624,E2 20003.624} C_VEL
LIN {X 0,Y 561.376,Z 421.253,A -85,B 0,C 180,E1 20000.651,E2 20000.651} C_VEL
LIN {X 0,Y 561.407,Z 421.298,A -85,B 0,C 180,E1 19997.304,E2 19997.304} C_VEL
LIN {X 0,Y 561.4,Z 421.248,A -85,B 0,C 180,E1 19994.228,E2 19994.228} C_VEL
LIN {X 0,Y 561.395,Z 421.279,A -85,B 0,C 180,E1 19990.883,E2 19990.883} C_VEL
LIN {X 0,Y 561.441,Z 421.257,A -85,B 0,C 180,E1 19987.676,E2 19987.676} C_VEL
LIN {X 0,Y 561.395,Z 421.265,A -85,B 0,C 180,E1 19984.495,E2 19984.495} C_VEL
LIN {X 0,Y 561.442,Z 421.269,A -85,B 0,C 180,E1 19981.225,E2 19981.225} C_VEL
LIN {X 0,Y 561.411,Z 421.251,A -85,B 0,C 180,E1 19977.959,E2 19977.959} C_VEL
LIN {X 0,Y 561.419,Z 421.295,A -85,B 0,C 180,E1 19974.481,E2 19974.481} C_VEL
LIN {X 0,Y 561.431,Z 421.241,A -85,B 0,C 180,E1 19971.279,E2 19971.279} C_VEL
LIN {X 0,Y 561.42,Z 421.299,A -85,B 0,C 180,E1 19967.973,E2 19967.973} C_VEL
LIN {X 0,Y 561.429,Z 421.243,A -85,B 0,C 180,E1 19964.717,E2 19964.717} C_VEL
LIN {X 0,Y 561.435,Z 421.277,A -85,B 0,C 180,E1 19961.302,E2 19961.302} C_VEL
LIN {X 0,Y 561.43,Z 421.273,A -85,B 0,C 180,E1 19957.927,E2 19957.927} C_VEL
LIN {X 0,Y 561.418,Z 421.248,A -85,B 0,C 180,E1 19954.694,E2 19954.694} C_VEL
LIN {X 0,Y 561.448,Z 421.431,A -85,B 0,C 180,E1 19952.336,E2 19952.336} C_VEL
LIN {X 0,Y 562.422,Z 424.249,A -85,B 0,C 180,E1 19952.071,E2 19952.071} C_VEL
LIN {X 0,Y 564.756,Z 426.827,A -85,B 0,C 180,E1 19951.558,E2 19951.558} C_VEL
LIN {X 0,Y 566.594,Z 428.047,A -85,B 0,C 180,E1 19951.184,E2 19951.184} C_VEL
LIN {X 0,Y 568.707,Z 431.588,A -85,B 0,C 180,E1 19950.708,E2 19950.708} C_VEL
LIN {X 0,Y 571.838,Z 434.431,A -85,B 0,C 180,E1 19950.081,E2 19950.081} C_VEL
LIN {X 0,Y 574.792,Z 438.512,A -85,B 0,C 180,E1 19949.472,E2 19949.472} C_VEL
LIN {X 0,Y 576.868,Z 440.559,A -85,B 0,C 180,E1 19949.074,E2 19949.074} C_VEL
LIN {X 0,Y 580.29,Z 444.925,A -85,B 0,C 180,E1 19948.411,E2 19948.411} C_VEL
LIN {X 0,Y 582.156,Z 447.164,A -85,B 0,C 180,E1 19948.061,E2 19948.061} C_VEL
LIN {X 0,Y 587.485,Z 453.774,A -85,B 0,C 180,E1 19947.087,E2 19947.087} C_VEL
LIN {X 0,Y 596.638,Z 465.769,A -85,B 0,C 180,E1 19945.497,E2 19945.497} C_VEL
LIN {X 0,Y 609.74,Z 484.146,A -85,B 0,C 180,E1 19943.38,E2 19943.38} C_VEL
LIN {X 0,Y 619.387,Z 498.754,A -85,B 0,C 180,E1 19941.921,E2 19941.921} C_VEL
LIN {X 0,Y 612.652,Z 712.627,A -85,B 0,C 180,E1 19938.841,E2 19938.841} C_VEL
LIN {X 0,Y 610.243,Z 792.846,A -85,B 0,C 180,E1 19937.705,E2 19937.705} C_VEL
LIN {X 0,Y 609.334,Z 800.551,A -85,B 0,C 180,E1 19937.667,E2 19937.667} C_VEL
LIN {X 0,Y 604.513,Z 821.189,A -85,B 0,C 180,E1 19937.813,E2 19937.813} C_VEL
LIN {X 0,Y 603.808,Z 827.797,A -85,B 0,C 180,E1 19937.773,E2 19937.773} C_VEL
LIN {X 0,Y 601.512,Z 896.456,A -85,B 0,C 180,E1 19936.782,E2 19936.782} C_VEL
LIN {X 0,Y 599.663,Z 924.651,A -85,B 0,C 180,E1 19936.238,E2 19936.238} C_VEL
LIN {X 0,Y 597.461,Z 949.163,A -85,B 0,C 180,E1 19935.595,E2 19935.595} C_VEL
LIN {X 0,Y 595.311,Z 969.725,A -85,B 0,C 180,E1 19934.934,E2 19934.934} C_VEL
LIN {X 0,Y 592.843,Z 990.297,A -85,B 0,C 180,E1 19934.153,E2 19934.153} C_VEL
LIN {X 0,Y 590.135,Z 1011.004,A -85,B 0,C 180,E1 19933.233,E2 19933.233} C_VEL
LIN {X 0,Y 586.69,Z 1034.919,A -85,B 0,C 180,E1 19932.006,E2 19932.006} C_VEL
LIN {X 0,Y 582.809,Z 1058.732,A -85,B 0,C 180,E1 19930.56,E2 19930.56} C_VEL
LIN {X 0,Y 579.66,Z 1077.313,A -85,B 0,C 180,E1 19929.278,E2 19929.278} C_VEL
LIN {X 0,Y 576.615,Z 1094.735,A -85,B 0,C 180,E1 19927.933,E2 19927.933} C_VEL
LIN {X 0,Y 573.361,Z 1113.001,A -85,B 0,C 180,E1 19926.367,E2 19926.367} C_VEL
LIN {X 0,Y 569.463,Z 1134.683,A -85,B 0,C 180,E1 19924.266,E2 19924.266} C_VEL
LIN {X 0,Y 566.27,Z 1152.536,A -85,B 0,C 180,E1 19922.287,E2 19922.287} C_VEL
LIN {X 0,Y 563.664,Z 1167.494,A -85,B 0,C 180,E1 19920.444,E2 19920.444} C_VEL
LIN {X 0,Y 561.095,Z 1183.003,A -85,B 0,C 180,E1 19918.318,E2 19918.318} C_VEL
LIN {X 0,Y 558.462,Z 1199.921,A -85,B 0,C 180,E1 19915.678,E2 19915.678} C_VEL
LIN {X 0,Y 556.613,Z 1212.865,A -85,B 0,C 180,E1 19913.371,E2 19913.371} C_VEL
LIN {X 0,Y 555.171,Z 1224.17,A -85,B 0,C 180,E1 19911.101,E2 19911.101} C_VEL
LIN {X 0,Y 553.857,Z 1236.272,A -85,B 0,C 180,E1 19908.31,E2 19908.31} C_VEL
LIN {X 0,Y 553.018,Z 1245.643,A -85,B 0,C 180,E1 19905.739,E2 19905.739} C_VEL
LIN {X 0,Y 552.523,Z 1252.609,A -85,B 0,C 180,E1 19903.503,E2 19903.503} C_VEL
LIN {X 0,Y 552.216,Z 1258.448,A -85,B 0,C 180,E1 19901.28,E2 19901.28} C_VEL
LIN {X 0,Y 552.016,Z 1263.439,A -85,B 0,C 180,E1 19898.964,E2 19898.964} C_VEL
LIN {X 0,Y 551.945,Z 1267.995,A -85,B 0,C 180,E1 19896.138,E2 19896.138} C_VEL
LIN {X 0,Y 551.913,Z 1270.575,A -85,B 0,C 180,E1 19893.534,E2 19893.534} C_VEL
LIN {X 0,Y 551.897,Z 1271.725,A -85,B 0,C 180,E1 19891.249,E2 19891.249} C_VEL
LIN {X 0,Y 551.866,Z 1271.837,A -85,B 0,C 180,E1 19889.173,E2 19889.173} C_VEL
LIN {X 0,Y 551.911,Z 1270.978,A -85,B 0,C 180,E1 19886.991,E2 19886.991} C_VEL
LIN {X 0,Y 551.923,Z 1269.039,A -85,B 0,C 180,E1 19884.702,E2 19884.702} C_VEL
LIN {X 0,Y 551.958,Z 1265.807,A -85,B 0,C 180,E1 19882.3,E2 19882.3} C_VEL
LIN {X 0,Y 552.148,Z 1260.598,A -85,B 0,C 180,E1 19879.524,E2 19879.524} C_VEL
LIN {X 0,Y 552.475,Z 1253.792,A -85,B 0,C 180,E1 19876.822,E2 19876.822} C_VEL
LIN {X 0,Y 552.944,Z 1246.668,A -85,B 0,C 180,E1 19874.481,E2 19874.481} C_VEL
LIN {X 0,Y 553.624,Z 1238.669,A -85,B 0,C 180,E1 19872.232,E2 19872.232} C_VEL
LIN {X 0,Y 554.751,Z 1228.04,A -85,B 0,C 180,E1 19869.647,E2 19869.647} C_VEL
LIN {X 0,Y 556.334,Z 1214.961,A -85,B 0,C 180,E1 19866.937,E2 19866.937} C_VEL
LIN {X 0,Y 558.075,Z 1202.363,A -85,B 0,C 180,E1 19864.651,E2 19864.651} C_VEL
LIN {X 0,Y 560.242,Z 1188.169,A -85,B 0,C 180,E1 19862.357,E2 19862.357} C_VEL
LIN {X 0,Y 563.203,Z 1170.359,A -85,B 0,C 180,E1 19859.838,E2 19859.838} C_VEL
LIN {X 0,Y 565.905,Z 1154.674,A -85,B 0,C 180,E1 19857.876,E2 19857.876} C_VEL
LIN {X 0,Y 568.712,Z 1138.777,A -85,B 0,C 180,E1 19856.084,E2 19856.084} C_VEL
LIN {X 0,Y 571.919,Z 1120.942,A -85,B 0,C 180,E1 19854.278,E2 19854.278} C_VEL
LIN {X 0,Y 576.079,Z 1097.766,A -85,B 0,C 180,E1 19852.221,E2 19852.221} C_VEL
LIN {X 0,Y 579.327,Z 1079.245,A -85,B 0,C 180,E1 19850.773,E2 19850.773} C_VEL
LIN {X 0,Y 582.446,Z 1060.847,A -85,B 0,C 180,E1 19849.488,E2 19849.488} C_VEL
LIN {X 0,Y 585.673,Z 1040.898,A -85,B 0,C 180,E1 19848.251,E2 19848.251} C_VEL
LIN {X 0,Y 589.386,Z 1016.623,A -85,B 0,C 180,E1 19846.941,E2 19846.941} C_VEL
LIN {X 0,Y 592.616,Z 992.157,A -85,B 0,C 180,E1 19845.833,E2 19845.833} C_VEL
LIN {X 0,Y 595.089,Z 971.702,A -85,B 0,C 180,E1 19845.046,E2 19845.046} C_VEL
LIN {X 0,Y 597.316,Z 950.549,A -85,B 0,C 180,E1 19844.356,E2 19844.356} C_VEL
LIN {X 0,Y 599.311,Z 928.641,A -85,B 0,C 180,E1 19843.77,E2 19843.77} C_VEL
LIN {X 0,Y 601.283,Z 901.412,A -85,B 0,C 180,E1 19843.206,E2 19843.206} C_VEL
LIN {X 0,Y 602.948,Z 856.059,A -85,B 0,C 180,E1 19842.537,E2 19842.537} C_VEL
LIN {X 0,Y 609.894,Z 635.794,A -85,B 0,C 180,E1 19839.393,E2 19839.393} C_VEL
LIN {X 0,Y 614.269,Z 502.597,A -85,B 0,C 180,E1 19837.443,E2 19837.443} C_VEL
LIN {X 0,Y 602.732,Z 485.403,A -85,B 0,C 180,E1 19835.641,E2 19835.641} C_VEL
LIN {X 0,Y 588.857,Z 466.13,A -85,B 0,C 180,E1 19833.291,E2 19833.291} C_VEL
LIN {X 0,Y 582.07,Z 457.472,A -85,B 0,C 180,E1 19832.06,E2 19832.06} C_VEL
LIN {X 0,Y 577.431,Z 451.771,A -85,B 0,C 180,E1 19831.182,E2 19831.182} C_VEL
LIN {X 0,Y 573.135,Z 446.509,A -85,B 0,C 180,E1 19830.336,E2 19830.336} C_VEL
LIN {X 0,Y 569.596,Z 442.264,A -85,B 0,C 180,E1 19829.614,E2 19829.614} C_VEL
LIN {X 0,Y 568.519,Z 440.848,A -85,B 0,C 180,E1 19829.386,E2 19829.386} C_VEL
LIN {X 0,Y 565.141,Z 437.335,A -85,B 0,C 180,E1 19828.68,E2 19828.68} C_VEL
LIN {X 0,Y 563.614,Z 434.928,A -85,B 0,C 180,E1 19828.331,E2 19828.331} C_VEL
LIN {X 0,Y 560.414,Z 432.049,A -85,B 0,C 180,E1 19827.639,E2 19827.639} C_VEL
LIN {X 0,Y 558.477,Z 428.741,A -85,B 0,C 180,E1 19827.165,E2 19827.165} C_VEL
LIN {X 0,Y 555.446,Z 426.601,A -85,B 0,C 180,E1 19826.487,E2 19826.487} C_VEL
LIN {X 0,Y 553.813,Z 423.683,A -85,B 0,C 180,E1 19826.06,E2 19826.06} C_VEL
LIN {X 0,Y 553.491,Z 422.234,A -85,B 0,C 180,E1 19825.924,E2 19825.924} C_VEL
LIN {X 0,Y 553.44,Z 422.295,A -85,B 0,C 180,E1 19822.745,E2 19822.745} C_VEL
LIN {X 0,Y 553.463,Z 422.242,A -85,B 0,C 180,E1 19819.416,E2 19819.416} C_VEL
LIN {X 0,Y 553.441,Z 422.261,A -85,B 0,C 180,E1 19816.37,E2 19816.37} C_VEL
LIN {X 0,Y 553.44,Z 422.266,A -85,B 0,C 180,E1 19812.946,E2 19812.946} C_VEL
LIN {X 0,Y 553.456,Z 422.24,A -85,B 0,C 180,E1 19809.883,E2 19809.883} C_VEL
LIN {X 0,Y 553.433,Z 422.281,A -85,B 0,C 180,E1 19806.64,E2 19806.64} C_VEL
LIN {X 0,Y 553.467,Z 422.233,A -85,B 0,C 180,E1 19803.522,E2 19803.522} C_VEL
LIN {X 0,Y 553.429,Z 422.291,A -85,B 0,C 180,E1 19800.311,E2 19800.311} C_VEL
LIN {X 0,Y 553.474,Z 422.23,A -85,B 0,C 180,E1 19797.204,E2 19797.204} C_VEL
LIN {X 0,Y 553.423,Z 422.293,A -85,B 0,C 180,E1 19793.985,E2 19793.985} C_VEL
LIN {X 0,Y 553.485,Z 422.227,A -85,B 0,C 180,E1 19790.853,E2 19790.853} C_VEL
LIN {X 0,Y 553.421,Z 422.294,A -85,B 0,C 180,E1 19787.584,E2 19787.584} C_VEL
LIN {X 0,Y 553.463,Z 422.233,A -85,B 0,C 180,E1 19784.328,E2 19784.328} C_VEL
LIN {X 0,Y 553.42,Z 422.269,A -85,B 0,C 180,E1 19781.24,E2 19781.24} C_VEL
LIN {X 0,Y 553.441,Z 422.257,A -85,B 0,C 180,E1 19777.927,E2 19777.927} C_VEL
LIN {X 0,Y 553.416,Z 422.245,A -85,B 0,C 180,E1 19774.989,E2 19774.989} C_VEL
LIN {X 0,Y 553.467,Z 422.35,A -85,B 0,C 180,E1 19774.534,E2 19774.534} C_VEL
LIN {X 0,Y 554.933,Z 426.002,A -85,B 0,C 180,E1 19773.746,E2 19773.746} C_VEL
LIN {X 0,Y 557.538,Z 428.802,A -85,B 0,C 180,E1 19773.132,E2 19773.132} C_VEL
LIN {X 0,Y 560.786,Z 432.651,A -85,B 0,C 180,E1 19772.381,E2 19772.381} C_VEL
LIN {X 0,Y 562.529,Z 434.902,A -85,B 0,C 180,E1 19771.985,E2 19771.985} C_VEL
LIN {X 0,Y 566.012,Z 439.041,A -85,B 0,C 180,E1 19771.224,E2 19771.224} C_VEL
LIN {X 0,Y 572.62,Z 447.528,A -85,B 0,C 180,E1 19769.837,E2 19769.837} C_VEL
LIN {X 0,Y 579.637,Z 456.489,A -85,B 0,C 180,E1 19768.458,E2 19768.458} C_VEL
LIN {X 0,Y 587.859,Z 467.519,A -85,B 0,C 180,E1 19766.937,E2 19766.937} C_VEL
LIN {X 0,Y 597.035,Z 480.123,A -85,B 0,C 180,E1 19765.348,E2 19765.348} C_VEL
LIN {X 0,Y 610.154,Z 499.512,A -85,B 0,C 180,E1 19763.233,E2 19763.233} C_VEL
LIN {X 0,Y 614.395,Z 506.311,A -85,B 0,C 180,E1 19762.58,E2 19762.58} C_VEL
LIN {X 0,Y 607.44,Z 717.742,A -85,B 0,C 180,E1 19759.517,E2 19759.517} C_VEL
LIN {X 0,Y 601.554,Z 903.248,A -85,B 0,C 180,E1 19756.868,E2 19756.868} C_VEL
LIN {X 0,Y 600.081,Z 927.044,A -85,B 0,C 180,E1 19756.434,E2 19756.434} C_VEL
LIN {X 0,Y 597.637,Z 955.837,A -85,B 0,C 180,E1 19755.72,E2 19755.72} C_VEL
LIN {X 0,Y 595.343,Z 977.865,A -85,B 0,C 180,E1 19755.025,E2 19755.025} C_VEL
LIN {X 0,Y 592.95,Z 998.03,A -85,B 0,C 180,E1 19754.27,E2 19754.27} C_VEL
LIN {X 0,Y 590.373,Z 1017.974,A -85,B 0,C 180,E1 19753.399,E2 19753.399} C_VEL
LIN {X 0,Y 587.433,Z 1038.467,A -85,B 0,C 180,E1 19752.377,E2 19752.377} C_VEL
LIN {X 0,Y 583.593,Z 1063.588,A -85,B 0,C 180,E1 19750.924,E2 19750.924} C_VEL
LIN {X 0,Y 580.041,Z 1084.791,A -85,B 0,C 180,E1 19749.495,E2 19749.495} C_VEL
LIN {X 0,Y 576.857,Z 1103.234,A -85,B 0,C 180,E1 19748.097,E2 19748.097} C_VEL
LIN {X 0,Y 573.916,Z 1119.867,A -85,B 0,C 180,E1 19746.691,E2 19746.691} C_VEL
LIN {X 0,Y 570.924,Z 1136.554,A -85,B 0,C 180,E1 19745.126,E2 19745.126} C_VEL
LIN {X 0,Y 567.651,Z 1154.93,A -85,B 0,C 180,E1 19743.207,E2 19743.207} C_VEL
LIN {X 0,Y 564.226,Z 1174.165,A -85,B 0,C 180,E1 19740.92,E2 19740.92} C_VEL
LIN {X 0,Y 561.764,Z 1188.861,A -85,B 0,C 180,E1 19738.951,E2 19738.951} C_VEL
LIN {X 0,Y 559.533,Z 1202.799,A -85,B 0,C 180,E1 19736.875,E2 19736.875} C_VEL
LIN {X 0,Y 557.232,Z 1218.402,A -85,B 0,C 180,E1 19734.258,E2 19734.258} C_VEL
LIN {X 0,Y 555.506,Z 1231.278,A -85,B 0,C 180,E1 19731.754,E2 19731.754} C_VEL
LIN {X 0,Y 554.387,Z 1241.079,A -85,B 0,C 180,E1 19729.597,E2 19729.597} C_VEL
LIN {X 0,Y 553.475,Z 1250.122,A -85,B 0,C 180,E1 19727.339,E2 19727.339} C_VEL
LIN {X 0,Y 552.776,Z 1258.992,A -85,B 0,C 180,E1 19724.773,E2 19724.773} C_VEL
LIN {X 0,Y 552.29,Z 1267.045,A -85,B 0,C 180,E1 19721.907,E2 19721.907} C_VEL
LIN {X 0,Y 552.034,Z 1272.301,A -85,B 0,C 180,E1 19719.589,E2 19719.589} C_VEL
LIN {X 0,Y 551.964,Z 1276.377,A -85,B 0,C 180,E1 19717.282,E2 19717.282} C_VEL
LIN {X 0,Y 551.921,Z 1279.445,A -85,B 0,C 180,E1 19714.881,E2 19714.881} C_VEL
LIN {X 0,Y 551.91,Z 1281.55,A -85,B 0,C 180,E1 19712.073,E2 19712.073} C_VEL
LIN {X 0,Y 551.865,Z 1281.871,A -85,B 0,C 180,E1 19709.374,E2 19709.374} C_VEL
LIN {X 0,Y 551.91,Z 1281.081,A -85,B 0,C 180,E1 19707.193,E2 19707.193} C_VEL
LIN {X 0,Y 551.922,Z 1279.21,A -85,B 0,C 180,E1 19704.904,E2 19704.904} C_VEL
LIN {X 0,Y 551.96,Z 1276.207,A -85,B 0,C 180,E1 19702.608,E2 19702.608} C_VEL
LIN {X 0,Y 552.064,Z 1271.808,A -85,B 0,C 180,E1 19700.161,E2 19700.161} C_VEL
LIN {X 0,Y 552.404,Z 1264.858,A -85,B 0,C 180,E1 19697.24,E2 19697.24} C_VEL
LIN {X 0,Y 552.914,Z 1257.204,A -85,B 0,C 180,E1 19694.689,E2 19694.689} C_VEL
LIN {X 0,Y 553.554,Z 1249.288,A -85,B 0,C 180,E1 19692.441,E2 19692.441} C_VEL
LIN {X 0,Y 554.553,Z 1239.681,A -85,B 0,C 180,E1 19690.074,E2 19690.074} C_VEL
LIN {X 0,Y 556.147,Z 1226.422,A -85,B 0,C 180,E1 19687.258,E2 19687.258} C_VEL
LIN {X 0,Y 557.929,Z 1213.348,A -85,B 0,C 180,E1 19684.864,E2 19684.864} C_VEL
LIN {X 0,Y 559.863,Z 1200.658,A -85,B 0,C 180,E1 19682.791,E2 19682.791} C_VEL
LIN {X 0,Y 562.419,Z 1184.962,A -85,B 0,C 180,E1 19680.496,E2 19680.496} C_VEL
LIN {X 0,Y 565.661,Z 1166.124,A -85,B 0,C 180,E1 19678.092,E2 19678.092} C_VEL
LIN {X 0,Y 568.416,Z 1150.455,A -85,B 0,C 180,E1 19676.31,E2 19676.31} C_VEL
LIN {X 0,Y 571.345,Z 1134.172,A -85,B 0,C 180,E1 19674.64,E2 19674.64} C_VEL
LIN {X 0,Y 574.573,Z 1116.142,A -85,B 0,C 180,E1 19672.977,E2 19672.977} C_VEL
LIN {X 0,Y 578.813,Z 1091.882,A -85,B 0,C 180,E1 19671.021,E2 19671.021} C_VEL
LIN {X 0,Y 582.107,Z 1072.235,A -85,B 0,C 180,E1 19669.64,E2 19669.64} C_VEL
LIN {X 0,Y 585.247,Z 1052.668,A -85,B 0,C 180,E1 19668.419,E2 19668.419} C_VEL
LIN {X 0,Y 588.315,Z 1032.357,A -85,B 0,C 180,E1 19667.301,E2 19667.301} C_VEL
LIN {X 0,Y 591.881,Z 1006.894,A -85,B 0,C 180,E1 19666.093,E2 19666.093} C_VEL
LIN {X 0,Y 594.863,Z 982.143,A -85,B 0,C 180,E1 19665.125,E2 19665.125} C_VEL
LIN {X 0,Y 597.123,Z 960.807,A -85,B 0,C 180,E1 19664.425,E2 19664.425} C_VEL
LIN {X 0,Y 599.073,Z 939.648,A -85,B 0,C 180,E1 19663.855,E2 19663.855} C_VEL
LIN {X 0,Y 600.771,Z 916.998,A -85,B 0,C 180,E1 19663.367,E2 19663.367} C_VEL
LIN {X 0,Y 602.373,Z 882.282,A -85,B 0,C 180,E1 19662.82,E2 19662.82} C_VEL
LIN {X 0,Y 609.366,Z 657.584,A -85,B 0,C 180,E1 19659.62,E2 19659.62} C_VEL
LIN {X 0,Y 614.327,Z 505.948,A -85,B 0,C 180,E1 19657.407,E2 19657.407} C_VEL
LIN {X 0,Y 603.306,Z 489.251,A -85,B 0,C 180,E1 19655.689,E2 19655.689} C_VEL
LIN {X 0,Y 590.609,Z 471.167,A -85,B 0,C 180,E1 19653.557,E2 19653.557} C_VEL
LIN {X 0,Y 581.437,Z 458.947,A -85,B 0,C 180,E1 19651.896,E2 19651.896} C_VEL
LIN {X 0,Y 574.128,Z 449.438,A -85,B 0,C 180,E1 19650.48,E2 19650.48} C_VEL
LIN {X 0,Y 569.706,Z 443.819,A -85,B 0,C 180,E1 19649.579,E2 19649.579} C_VEL
LIN {X 0,Y 565.947,Z 438.978,A -85,B 0,C 180,E1 19648.78,E2 19648.78} C_VEL
LIN {X 0,Y 562.465,Z 434.77,A -85,B 0,C 180,E1 19648.019,E2 19648.019} C_VEL
LIN {X 0,Y 560.925,Z 432.778,A -85,B 0,C 180,E1 19647.669,E2 19647.669} C_VEL
LIN {X 0,Y 557.657,Z 428.994,A -85,B 0,C 180,E1 19646.92,E2 19646.92} C_VEL
LIN {X 0,Y 556.456,Z 427.578,A -85,B 0,C 180,E1 19646.636,E2 19646.636} C_VEL
LIN {X 0,Y 554.338,Z 424.954,A -85,B 0,C 180,E1 19646.067,E2 19646.067} C_VEL
LIN {X 0,Y 553.445,Z 422.239,A -85,B 0,C 180,E1 19645.467,E2 19645.467} C_VEL
LIN {X 0,Y 553.457,Z 422.284,A -85,B 0,C 180,E1 19642.408,E2 19642.408} C_VEL
LIN {X 0,Y 553.444,Z 422.253,A -85,B 0,C 180,E1 19639.087,E2 19639.087} C_VEL
LIN {X 0,Y 553.492,Z 422.24,A -85,B 0,C 180,E1 19635.938,E2 19635.938} C_VEL
LIN {X 0,Y 553.45,Z 422.281,A -85,B 0,C 180,E1 19632.684,E2 19632.684} C_VEL
LIN {X 0,Y 553.498,Z 422.226,A -85,B 0,C 180,E1 19629.462,E2 19629.462} C_VEL
LIN {X 0,Y 553.464,Z 422.289,A -85,B 0,C 180,E1 19626.223,E2 19626.223} C_VEL
LIN {X 0,Y 553.47,Z 422.228,A -85,B 0,C 180,E1 19622.796,E2 19622.796} C_VEL
LIN {X 0,Y 553.505,Z 422.279,A -85,B 0,C 180,E1 19619.482,E2 19619.482} C_VEL
LIN {X 0,Y 553.466,Z 422.233,A -85,B 0,C 180,E1 19616.167,E2 19616.167} C_VEL
LIN {X 0,Y 553.506,Z 422.264,A -85,B 0,C 180,E1 19612.84,E2 19612.84} C_VEL
LIN {X 0,Y 553.494,Z 422.249,A -85,B 0,C 180,E1 19609.382,E2 19609.382} C_VEL
LIN {X 0,Y 553.478,Z 422.242,A -85,B 0,C 180,E1 19606.097,E2 19606.097} C_VEL
LIN {X 0,Y 553.493,Z 422.279,A -85,B 0,C 180,E1 19602.766,E2 19602.766} C_VEL
LIN {X 0,Y 553.495,Z 422.232,A -85,B 0,C 180,E1 19599.354,E2 19599.354} C_VEL
LIN {X 0,Y 553.495,Z 422.258,A -85,B 0,C 180,E1 19596.017,E2 19596.017} C_VEL
LIN {X 0,Y 553.514,Z 422.393,A -85,B 0,C 180,E1 19593.926,E2 19593.926} C_VEL
LIN {X 0,Y 554.494,Z 425.239,A -85,B 0,C 180,E1 19593.637,E2 19593.637} C_VEL
LIN {X 0,Y 556.993,Z 427.926,A -85,B 0,C 180,E1 19593.046,E2 19593.046} C_VEL
LIN {X 0,Y 558.799,Z 429.089,A -85,B 0,C 180,E1 19592.65,E2 19592.65} C_VEL
LIN {X 0,Y 560.945,Z 432.71,A -85,B 0,C 180,E1 19592.13,E2 19592.13} C_VEL
LIN {X 0,Y 564.066,Z 435.426,A -85,B 0,C 180,E1 19591.463,E2 19591.463} C_VEL
LIN {X 0,Y 566.882,Z 439.424,A -85,B 0,C 180,E1 19590.839,E2 19590.839} C_VEL
LIN {X 0,Y 569.324,Z 441.761,A -85,B 0,C 180,E1 19590.341,E2 19590.341} C_VEL
LIN {X 0,Y 572.726,Z 446.1,A -85,B 0,C 180,E1 19589.64,E2 19589.64} C_VEL
LIN {X 0,Y 574.532,Z 448.182,A -85,B 0,C 180,E1 19589.283,E2 19589.283} C_VEL
LIN {X 0,Y 579.676,Z 454.552,A -85,B 0,C 180,E1 19588.287,E2 19588.287} C_VEL
LIN {X 0,Y 584.616,Z 460.66,A -85,B 0,C 180,E1 19587.372,E2 19587.372} C_VEL
LIN {X 0,Y 593.559,Z 472.538,A -85,B 0,C 180,E1 19585.79,E2 19585.79} C_VEL
LIN {X 0,Y 606.293,Z 490.545,A -85,B 0,C 180,E1 19583.697,E2 19583.697} C_VEL
LIN {X 0,Y 614.33,Z 502.895,A -85,B 0,C 180,E1 19582.451,E2 19582.451} C_VEL
LIN {X 0,Y 607.176,Z 719.82,A -85,B 0,C 180,E1 19579.31,E2 19579.31} C_VEL
LIN {X 0,Y 603.808,Z 827.797,A -85,B 0,C 180,E1 19577.773,E2 19577.773} C_VEL
LIN {X 0,Y 602.902,Z 835.499,A -85,B 0,C 180,E1 19577.734,E2 19577.734} C_VEL
LIN {X 0,Y 598.051,Z 856.127,A -85,B 0,C 180,E1 19577.886,E2 19577.886} C_VEL
LIN {X 0,Y 597.341,Z 862.735,A -85,B 0,C 180,E1 19577.845,E2 19577.845} C_VEL
LIN {X 0,Y 595.71,Z 903.326,A -85,B 0,C 180,E1 19577.235,E2 19577.235} C_VEL
LIN {X 0,Y 593.69,Z 929.579,A -85,B 0,C 180,E1 19576.68,E2 19576.68} C_VEL
LIN {X 0,Y 591.664,Z 951.003,A -85,B 0,C 180,E1 19576.102,E2 19576.102} C_VEL
LIN {X 0,Y 589.436,Z 971.308,A -85,B 0,C 180,E1 19575.437,E2 19575.437} C_VEL
LIN {X 0,Y 586.875,Z 991.683,A -85,B 0,C 180,E1 19574.653,E2 19574.653} C_VEL
LIN {X 0,Y 583.655,Z 1015.19,A -85,B 0,C 180,E1 19573.588,E2 19573.588} C_VEL
LIN {X 0,Y 579.629,Z 1040.688,A -85,B 0,C 180,E1 19572.216,E2 19572.216} C_VEL
LIN {X 0,Y 576.287,Z 1060.449,A -85,B 0,C 180,E1 19570.986,E2 19570.986} C_VEL
LIN {X 0,Y 573.148,Z 1078.144,A -85,B 0,C 180,E1 19569.747,E2 19569.747} C_VEL
LIN {X 0,Y 569.963,Z 1095.499,A -85,B 0,C 180,E1 19568.392,E2 19568.392} C_VEL
LIN {X 0,Y 566.446,Z 1114.263,A -85,B 0,C 180,E1 19566.757,E2 19566.757} C_VEL
LIN {X 0,Y 562.223,Z 1136.358,A -85,B 0,C 180,E1 19564.566,E2 19564.566} C_VEL
LIN {X 0,Y 559.094,Z 1153.003,A -85,B 0,C 180,E1 19562.692,E2 19562.692} C_VEL
LIN {X 0,Y 556.334,Z 1168.023,A -85,B 0,C 180,E1 19560.814,E2 19560.814} C_VEL
LIN {X 0,Y 553.443,Z 1184.683,A -85,B 0,C 180,E1 19558.489,E2 19558.489} C_VEL
LIN {X 0,Y 550.81,Z 1200.558,A -85,B 0,C 180,E1 19555.946,E2 19555.946} C_VEL
LIN {X 0,Y 548.965,Z 1212.754,A -85,B 0,C 180,E1 19553.739,E2 19553.739} C_VEL
LIN {X 0,Y 547.477,Z 1223.59,A -85,B 0,C 180,E1 19551.539,E2 19551.539} C_VEL
LIN {X 0,Y 546.131,Z 1234.996,A -85,B 0,C 180,E1 19548.911,E2 19548.911} C_VEL
LIN {X 0,Y 545.138,Z 1245.292,A -85,B 0,C 180,E1 19546.081,E2 19546.081} C_VEL
LIN {X 0,Y 544.57,Z 1252.456,A -85,B 0,C 180,E1 19543.759,E2 19543.759} C_VEL
LIN {X 0,Y 544.26,Z 1258.195,A -85,B 0,C 180,E1 19541.554,E2 19541.554} C_VEL
LIN {X 0,Y 544.022,Z 1263.025,A -85,B 0,C 180,E1 19539.311,E2 19539.311} C_VEL
LIN {X 0,Y 543.957,Z 1267.095,A -85,B 0,C 180,E1 19536.865,E2 19536.865} C_VEL
LIN {X 0,Y 543.917,Z 1270.303,A -85,B 0,C 180,E1 19534.009,E2 19534.009} C_VEL
LIN {X 0,Y 543.903,Z 1271.703,A -85,B 0,C 180,E1 19531.372,E2 19531.372} C_VEL
LIN {X 0,Y 543.866,Z 1271.837,A -85,B 0,C 180,E1 19529.16,E2 19529.16} C_VEL
LIN {X 0,Y 543.912,Z 1270.978,A -85,B 0,C 180,E1 19526.947,E2 19526.947} C_VEL
LIN {X 0,Y 543.924,Z 1269.036,A -85,B 0,C 180,E1 19524.624,E2 19524.624} C_VEL
LIN {X 0,Y 543.959,Z 1265.963,A -85,B 0,C 180,E1 19522.292,E2 19522.292} C_VEL
LIN {X 0,Y 544.14,Z 1261.137,A -85,B 0,C 180,E1 19519.629,E2 19519.629} C_VEL
LIN {X 0,Y 544.504,Z 1254.056,A -85,B 0,C 180,E1 19516.721,E2 19516.721} C_VEL
LIN {X 0,Y 544.995,Z 1247.018,A -85,B 0,C 180,E1 19514.358,E2 19514.358} C_VEL
LIN {X 0,Y 545.72,Z 1239.07,A -85,B 0,C 180,E1 19512.076,E2 19512.076} C_VEL
LIN {X 0,Y 546.788,Z 1229.427,A -85,B 0,C 180,E1 19509.673,E2 19509.673} C_VEL
LIN {X 0,Y 548.581,Z 1215.528,A -85,B 0,C 180,E1 19506.706,E2 19506.706} C_VEL
LIN {X 0,Y 550.419,Z 1202.991,A -85,B 0,C 180,E1 19504.388,E2 19504.388} C_VEL
LIN {X 0,Y 552.49,Z 1190.045,A -85,B 0,C 180,E1 19502.251,E2 19502.251} C_VEL
LIN {X 0,Y 555.476,Z 1173.169,A -85,B 0,C 180,E1 19499.772,E2 19499.772} C_VEL
LIN {X 0,Y 558.756,Z 1154.883,A -85,B 0,C 180,E1 19497.443,E2 19497.443} C_VEL
LIN {X 0,Y 561.735,Z 1138.907,A -85,B 0,C 180,E1 19495.621,E2 19495.621} C_VEL
LIN {X 0,Y 565.275,Z 1120.285,A -85,B 0,C 180,E1 19493.717,E2 19493.717} C_VEL
LIN {X 0,Y 569.57,Z 1097.672,A -85,B 0,C 180,E1 19491.695,E2 19491.695} C_VEL
LIN {X 0,Y 572.953,Z 1079.253,A -85,B 0,C 180,E1 19490.244,E2 19490.244} C_VEL
LIN {X 0,Y 576.076,Z 1061.654,A -85,B 0,C 180,E1 19489.004,E2 19489.004} C_VEL
LIN {X 0,Y 579.245,Z 1042.898,A -85,B 0,C 180,E1 19487.824,E2 19487.824} C_VEL
LIN {X 0,Y 582.608,Z 1021.758,A -85,B 0,C 180,E1 19486.653,E2 19486.653} C_VEL
LIN {X 0,Y 586.486,Z 994.793,A -85,B 0,C 180,E1 19485.386,E2 19485.386} C_VEL
LIN {X 0,Y 589.281,Z 972.657,A -85,B 0,C 180,E1 19484.521,E2 19484.521} C_VEL
LIN {X 0,Y 591.618,Z 951.406,A -85,B 0,C 180,E1 19483.82,E2 19483.82} C_VEL
LIN {X 0,Y 593.643,Z 930.136,A -85,B 0,C 180,E1 19483.244,E2 19483.244} C_VEL
LIN {X 0,Y 595.484,Z 906.272,A -85,B 0,C 180,E1 19482.732,E2 19482.732} C_VEL
LIN {X 0,Y 597.111,Z 870.101,A -85,B 0,C 180,E1 19482.17,E2 19482.17} C_VEL
LIN {X 0,Y 604.44,Z 647.285,A -85,B 0,C 180,E1 19478.971,E2 19478.971} C_VEL
LIN {X 0,Y 609.264,Z 506.713,A -85,B 0,C 180,E1 19476.903,E2 19476.903} C_VEL
LIN {X 0,Y 597.336,Z 488.848,A -85,B 0,C 180,E1 19474.982,E2 19474.982} C_VEL
LIN {X 0,Y 584.883,Z 471.664,A -85,B 0,C 180,E1 19472.815,E2 19472.815} C_VEL
LIN {X 0,Y 579.24,Z 464.362,A -85,B 0,C 180,E1 19471.769,E2 19471.769} C_VEL
LIN {X 0,Y 574.186,Z 458.181,A -85,B 0,C 180,E1 19470.796,E2 19470.796} C_VEL
LIN {X 0,Y 570.39,Z 453.455,A -85,B 0,C 180,E1 19470.032,E2 19470.032} C_VEL
LIN {X 0,Y 566.686,Z 448.83,A -85,B 0,C 180,E1 19469.259,E2 19469.259} C_VEL
LIN {X 0,Y 562.289,Z 443.909,A -85,B 0,C 180,E1 19468.317,E2 19468.317} C_VEL
LIN {X 0,Y 560.959,Z 442.049,A -85,B 0,C 180,E1 19468.014,E2 19468.014} C_VEL
LIN {X 0,Y 557.525,Z 438.507,A -85,B 0,C 180,E1 19467.244,E2 19467.244} C_VEL
LIN {X 0,Y 556.081,Z 436.142,A -85,B 0,C 180,E1 19466.887,E2 19466.887} C_VEL
LIN {X 0,Y 552.916,Z 433.507,A -85,B 0,C 180,E1 19466.155,E2 19466.155} C_VEL
LIN {X 0,Y 550.823,Z 429.788,A -85,B 0,C 180,E1 19465.597,E2 19465.597} C_VEL
LIN {X 0,Y 547.647,Z 427.764,A -85,B 0,C 180,E1 19464.83,E2 19464.83} C_VEL
LIN {X 0,Y 545.937,Z 424.943,A -85,B 0,C 180,E1 19464.351,E2 19464.351} C_VEL
LIN {X 0,Y 545.547,Z 423.234,A -85,B 0,C 180,E1 19464.182,E2 19464.182} C_VEL
LIN {X 0,Y 545.491,Z 423.23,A -85,B 0,C 180,E1 19460.943,E2 19460.943} C_VEL
LIN {X 0,Y 545.559,Z 423.276,A -85,B 0,C 180,E1 19457.646,E2 19457.646} C_VEL
LIN {X 0,Y 545.489,Z 423.222,A -85,B 0,C 180,E1 19454.436,E2 19454.436} C_VEL
LIN {X 0,Y 545.521,Z 423.267,A -85,B 0,C 180,E1 19451.096,E2 19451.096} C_VEL
LIN {X 0,Y 545.499,Z 423.226,A -85,B 0,C 180,E1 19448.008,E2 19448.008} C_VEL
LIN {X 0,Y 545.496,Z 423.252,A -85,B 0,C 180,E1 19444.626,E2 19444.626} C_VEL
LIN {X 0,Y 545.54,Z 423.234,A -85,B 0,C 180,E1 19441.365,E2 19441.365} C_VEL
LIN {X 0,Y 545.485,Z 423.244,A -85,B 0,C 180,E1 19438.214,E2 19438.214} C_VEL
LIN {X 0,Y 545.549,Z 423.243,A -85,B 0,C 180,E1 19434.953,E2 19434.953} C_VEL
LIN {X 0,Y 545.478,Z 423.235,A -85,B 0,C 180,E1 19431.78,E2 19431.78} C_VEL
LIN {X 0,Y 545.528,Z 423.262,A -85,B 0,C 180,E1 19428.476,E2 19428.476} C_VEL
LIN {X 0,Y 545.477,Z 423.226,A -85,B 0,C 180,E1 19425.41,E2 19425.41} C_VEL
LIN {X 0,Y 545.505,Z 423.277,A -85,B 0,C 180,E1 19422.028,E2 19422.028} C_VEL
LIN {X 0,Y 545.488,Z 423.224,A -85,B 0,C 180,E1 19418.944,E2 19418.944} C_VEL
LIN {X 0,Y 545.559,Z 423.419,A -85,B 0,C 180,E1 19416.129,E2 19416.129} C_VEL
LIN {X 0,Y 546.277,Z 425.85,A -85,B 0,C 180,E1 19415.651,E2 19415.651} C_VEL
LIN {X 0,Y 548.386,Z 428.471,A -85,B 0,C 180,E1 19415.09,E2 19415.09} C_VEL
LIN {X 0,Y 550.242,Z 429.959,A -85,B 0,C 180,E1 19414.634,E2 19414.634} C_VEL
LIN {X 0,Y 554.383,Z 435.036,A -85,B 0,C 180,E1 19413.603,E2 19413.603} C_VEL
LIN {X 0,Y 558.807,Z 440.201,A -85,B 0,C 180,E1 19412.564,E2 19412.564} C_VEL
LIN {X 0,Y 563.126,Z 445.794,A -85,B 0,C 180,E1 19411.584,E2 19411.584} C_VEL
LIN {X 0,Y 565.032,Z 448.149,A -85,B 0,C 180,E1 19411.169,E2 19411.169} C_VEL
LIN {X 0,Y 573.664,Z 459.197,A -85,B 0,C 180,E1 19409.377,E2 19409.377} C_VEL
LIN {X 0,Y 584.15,Z 473.195,A -85,B 0,C 180,E1 19407.372,E2 19407.372} C_VEL
LIN {X 0,Y 594.797,Z 488.204,A -85,B 0,C 180,E1 19405.492,E2 19405.492} C_VEL
LIN {X 0,Y 606.687,Z 505.91,A -85,B 0,C 180,E1 19403.548,E2 19403.548} C_VEL
LIN {X 0,Y 609.39,Z 510.421,A -85,B 0,C 180,E1 19403.119,E2 19403.119} C_VEL
LIN {X 0,Y 601.979,Z 725.763,A -85,B 0,C 180,E1 19399.983,E2 19399.983} C_VEL
LIN {X 0,Y 596.085,Z 903.229,A -85,B 0,C 180,E1 19397.43,E2 19397.43} C_VEL
LIN {X 0,Y 594.536,Z 927.281,A -85,B 0,C 180,E1 19396.99,E2 19396.99} C_VEL
LIN {X 0,Y 591.994,Z 955.965,A -85,B 0,C 180,E1 19396.274,E2 19396.274} C_VEL
LIN {X 0,Y 589.625,Z 977.776,A -85,B 0,C 180,E1 19395.584,E2 19395.584} C_VEL
LIN {X 0,Y 587.139,Z 997.94,A -85,B 0,C 180,E1 19394.826,E2 19394.826} C_VEL
LIN {X 0,Y 584.426,Z 1018.003,A -85,B 0,C 180,E1 19393.946,E2 19393.946} C_VEL
LIN {X 0,Y 581.365,Z 1038.423,A -85,B 0,C 180,E1 19392.922,E2 19392.922} C_VEL
LIN {X 0,Y 577.398,Z 1063.29,A -85,B 0,C 180,E1 19391.475,E2 19391.475} C_VEL
LIN {X 0,Y 573.647,Z 1084.7,A -85,B 0,C 180,E1 19390.023,E2 19390.023} C_VEL
LIN {X 0,Y 570.307,Z 1103.142,A -85,B 0,C 180,E1 19388.614,E2 19388.614} C_VEL
LIN {X 0,Y 567.164,Z 1120.129,A -85,B 0,C 180,E1 19387.168,E2 19387.168} C_VEL
LIN {X 0,Y 564.045,Z 1136.816,A -85,B 0,C 180,E1 19385.59,E2 19385.59} C_VEL
LIN {X 0,Y 560.387,Z 1156.412,A -85,B 0,C 180,E1 19383.515,E2 19383.515} C_VEL
LIN {X 0,Y 556.874,Z 1175.008,A -85,B 0,C 180,E1 19381.254,E2 19381.254} C_VEL
LIN {X 0,Y 554.282,Z 1189.629,A -85,B 0,C 180,E1 19379.261,E2 19379.261} C_VEL
LIN {X 0,Y 551.949,Z 1203.497,A -85,B 0,C 180,E1 19377.158,E2 19377.158} C_VEL
LIN {X 0,Y 549.43,Z 1219.569,A -85,B 0,C 180,E1 19374.396,E2 19374.396} C_VEL
LIN {X 0,Y 547.702,Z 1231.802,A -85,B 0,C 180,E1 19371.965,E2 19371.965} C_VEL
LIN {X 0,Y 546.527,Z 1241.537,A -85,B 0,C 180,E1 19369.779,E2 19369.779} C_VEL
LIN {X 0,Y 545.523,Z 1250.931,A -85,B 0,C 180,E1 19367.379,E2 19367.379} C_VEL
LIN {X 0,Y 544.73,Z 1260.321,A -85,B 0,C 180,E1 19364.561,E2 19364.561} C_VEL
LIN {X 0,Y 544.306,Z 1267.3,A -85,B 0,C 180,E1 19361.977,E2 19361.977} C_VEL
LIN {X 0,Y 544.053,Z 1272.298,A -85,B 0,C 180,E1 19359.731,E2 19359.731} C_VEL
LIN {X 0,Y 543.962,Z 1276.374,A -85,B 0,C 180,E1 19357.389,E2 19357.389} C_VEL
LIN {X 0,Y 543.923,Z 1279.328,A -85,B 0,C 180,E1 19355.059,E2 19355.059} C_VEL
LIN {X 0,Y 543.907,Z 1281.288,A -85,B 0,C 180,E1 19352.526,E2 19352.526} C_VEL
LIN {X 0,Y 543.878,Z 1281.938,A -85,B 0,C 180,E1 19349.681,E2 19349.681} C_VEL
LIN {X 0,Y 543.91,Z 1281.081,A -85,B 0,C 180,E1 19347.152,E2 19347.152} C_VEL
LIN {X 0,Y 543.923,Z 1279.207,A -85,B 0,C 180,E1 19344.829,E2 19344.829} C_VEL
LIN {X 0,Y 543.959,Z 1276.204,A -85,B 0,C 180,E1 19342.498,E2 19342.498} C_VEL
LIN {X 0,Y 544.079,Z 1271.931,A -85,B 0,C 180,E1 19340.08,E2 19340.08} C_VEL
LIN {X 0,Y 544.431,Z 1265.161,A -85,B 0,C 180,E1 19337.158,E2 19337.158} C_VEL
LIN {X 0,Y 544.986,Z 1257.203,A -85,B 0,C 180,E1 19334.46,E2 19334.46} C_VEL
LIN {X 0,Y 545.692,Z 1249.287,A -85,B 0,C 180,E1 19332.179,E2 19332.179} C_VEL
LIN {X 0,Y 546.774,Z 1239.525,A -85,B 0,C 180,E1 19329.74,E2 19329.74} C_VEL
LIN {X 0,Y 548.54,Z 1225.847,A -85,B 0,C 180,E1 19326.811,E2 19326.811} C_VEL
LIN {X 0,Y 550.362,Z 1213.345,A -85,B 0,C 180,E1 19324.494,E2 19324.494} C_VEL
LIN {X 0,Y 552.391,Z 1200.656,A -85,B 0,C 180,E1 19322.392,E2 19322.392} C_VEL
LIN {X 0,Y 555.181,Z 1184.693,A -85,B 0,C 180,E1 19320.031,E2 19320.031} C_VEL
LIN {X 0,Y 558.539,Z 1166.122,A -85,B 0,C 180,E1 19317.636,E2 19317.636} C_VEL
LIN {X 0,Y 561.482,Z 1150.273,A -85,B 0,C 180,E1 19315.815,E2 19315.815} C_VEL
LIN {X 0,Y 564.589,Z 1133.8,A -85,B 0,C 180,E1 19314.11,E2 19314.11} C_VEL
LIN {X 0,Y 568.227,Z 1114.424,A -85,B 0,C 180,E1 19312.321,E2 19312.321} C_VEL
LIN {X 0,Y 572.47,Z 1091.24,A -85,B 0,C 180,E1 19310.457,E2 19310.457} C_VEL
LIN {X 0,Y 575.823,Z 1072.144,A -85,B 0,C 180,E1 19309.106,E2 19309.106} C_VEL
LIN {X 0,Y 578.969,Z 1053.39,A -85,B 0,C 180,E1 19307.925,E2 19307.925} C_VEL
LIN {X 0,Y 582.145,Z 1033.275,A -85,B 0,C 180,E1 19306.805,E2 19306.805} C_VEL
LIN {X 0,Y 585.864,Z 1008.064,A -85,B 0,C 180,E1 19305.592,E2 19305.592} C_VEL
LIN {X 0,Y 589.046,Z 982.795,A -85,B 0,C 180,E1 19304.594,E2 19304.594} C_VEL
LIN {X 0,Y 591.432,Z 961.238,A -85,B 0,C 180,E1 19303.881,E2 19303.881} C_VEL
LIN {X 0,Y 593.453,Z 940.211,A -85,B 0,C 180,E1 19303.309,E2 19303.309} C_VEL
LIN {X 0,Y 595.178,Z 918.209,A -85,B 0,C 180,E1 19302.83,E2 19302.83} C_VEL
LIN {X 0,Y 596.706,Z 889.577,A -85,B 0,C 180,E1 19302.359,E2 19302.359} C_VEL
LIN {X 0,Y 603.99,Z 665.505,A -85,B 0,C 180,E1 19299.148,E2 19299.148} C_VEL
LIN {X 0,Y 609.325,Z 510.075,A -85,B 0,C 180,E1 19296.869,E2 19296.869} C_VEL
LIN {X 0,Y 599.647,Z 495.289,A -85,B 0,C 180,E1 19295.324,E2 19295.324} C_VEL
LIN {X 0,Y 587.452,Z 477.747,A -85,B 0,C 180,E1 19293.235,E2 19293.235} C_VEL
LIN {X 0,Y 578.261,Z 465.383,A -85,B 0,C 180,E1 19291.538,E2 19291.538} C_VEL
LIN {X 0,Y 571.15,Z 456.05,A -85,B 0,C 180,E1 19290.133,E2 19290.133} C_VEL
LIN {X 0,Y 566.781,Z 450.451,A -85,B 0,C 180,E1 19289.224,E2 19289.224} C_VEL
LIN {X 0,Y 563.167,Z 445.827,A -85,B 0,C 180,E1 19288.442,E2 19288.442} C_VEL
LIN {X 0,Y 559.547,Z 441.166,A -85,B 0,C 180,E1 19287.627,E2 19287.627} C_VEL
LIN {X 0,Y 555.001,Z 435.721,A -85,B 0,C 180,E1 19286.567,E2 19286.567} C_VEL
LIN {X 0,Y 550.066,Z 429.694,A -85,B 0,C 180,E1 19285.346,E2 19285.346} C_VEL
LIN {X 0,Y 546.892,Z 426.837,A -85,B 0,C 180,E1 19284.55,E2 19284.55} C_VEL
LIN {X 0,Y 545.874,Z 424.729,A -85,B 0,C 180,E1 19284.188,E2 19284.188} C_VEL
LIN {X 0,Y 545.555,Z 423.242,A -85,B 0,C 180,E1 19283.855,E2 19283.855} C_VEL
LIN {X 0,Y 545.497,Z 423.228,A -85,B 0,C 180,E1 19280.718,E2 19280.718} C_VEL
LIN {X 0,Y 545.536,Z 423.277,A -85,B 0,C 180,E1 19277.383,E2 19277.383} C_VEL
LIN {X 0,Y 545.527,Z 423.222,A -85,B 0,C 180,E1 19274.163,E2 19274.163} C_VEL
LIN {X 0,Y 545.517,Z 423.252,A -85,B 0,C 180,E1 19270.882,E2 19270.882} C_VEL
LIN {X 0,Y 545.565,Z 423.233,A -85,B 0,C 180,E1 19267.583,E2 19267.583} C_VEL
LIN {X 0,Y 545.519,Z 423.232,A -85,B 0,C 180,E1 19264.31,E2 19264.31} C_VEL
LIN {X 0,Y 545.554,Z 423.254,A -85,B 0,C 180,E1 19260.945,E2 19260.945} C_VEL
LIN {X 0,Y 545.552,Z 423.216,A -85,B 0,C 180,E1 19257.584,E2 19257.584} C_VEL
LIN {X 0,Y 545.535,Z 423.275,A -85,B 0,C 180,E1 19254.214,E2 19254.214} C_VEL
LIN {X 0,Y 545.554,Z 423.212,A -85,B 0,C 180,E1 19250.931,E2 19250.931} C_VEL
LIN {X 0,Y 545.558,Z 423.27,A -85,B 0,C 180,E1 19247.51,E2 19247.51} C_VEL
LIN {X 0,Y 545.545,Z 423.225,A -85,B 0,C 180,E1 19244.152,E2 19244.152} C_VEL
LIN {X 0,Y 545.547,Z 423.236,A -85,B 0,C 180,E1 19240.848,E2 19240.848} C_VEL
LIN {X 0,Y 545.561,Z 423.262,A -85,B 0,C 180,E1 19237.477,E2 19237.477} C_VEL
LIN {X 0,Y 545.568,Z 423.373,A -85,B 0,C 180,E1 19235.665,E2 19235.665} C_VEL
LIN {X 0,Y 546.554,Z 426.225,A -85,B 0,C 180,E1 19235.347,E2 19235.347} C_VEL
LIN {X 0,Y 548.994,Z 428.86,A -85,B 0,C 180,E1 19234.716,E2 19234.716} C_VEL
LIN {X 0,Y 551.003,Z 430.099,A -85,B 0,C 180,E1 19234.239,E2 19234.239} C_VEL
LIN {X 0,Y 553.021,Z 433.605,A -85,B 0,C 180,E1 19233.706,E2 19233.706} C_VEL
LIN {X 0,Y 556.485,Z 436.71,A -85,B 0,C 180,E1 19232.904,E2 19232.904} C_VEL
LIN {X 0,Y 559.27,Z 440.637,A -85,B 0,C 180,E1 19232.242,E2 19232.242} C_VEL
LIN {X 0,Y 561.715,Z 442.918,A -85,B 0,C 180,E1 19231.709,E2 19231.709} C_VEL
LIN {X 0,Y 565.077,Z 447.211,A -85,B 0,C 180,E1 19230.969,E2 19230.969} C_VEL
LIN {X 0,Y 566.829,Z 449.019,A -85,B 0,C 180,E1 19230.604,E2 19230.604} C_VEL
LIN {X 0,Y 570.667,Z 453.674,A -85,B 0,C 180,E1 19229.81,E2 19229.81} C_VEL
LIN {X 0,Y 577.209,Z 461.904,A -85,B 0,C 180,E1 19228.514,E2 19228.514} C_VEL
LIN {X 0,Y 583.42,Z 469.62,A -85,B 0,C 180,E1 19227.355,E2 19227.355} C_VEL
LIN {X 0,Y 594.672,Z 485.213,A -85,B 0,C 180,E1 19225.367,E2 19225.367} C_VEL
LIN {X 0,Y 606.072,Z 501.758,A -85,B 0,C 180,E1 19223.505,E2 19223.505} C_VEL
LIN {X 0,Y 609.323,Z 507.106,A -85,B 0,C 180,E1 19222.989,E2 19222.989} C_VEL
LIN {X 0,Y 601.864,Z 723.317,A -85,B 0,C 180,E1 19219.84,E2 19219.84} C_VEL
LIN {X 0,Y 597.341,Z 862.735,A -85,B 0,C 180,E1 19217.845,E2 19217.845} C_VEL
LIN {X 0,Y 596.426,Z 870.436,A -85,B 0,C 180,E1 19217.809,E2 19217.809} C_VEL
LIN {X 0,Y 591.413,Z 891.034,A -85,B 0,C 180,E1 19217.953,E2 19217.953} C_VEL
LIN {X 0,Y 590.599,Z 897.624,A -85,B 0,C 180,E1 19217.901,E2 19217.901} C_VEL
LIN {X 0,Y 588.46,Z 926.891,A -85,B 0,C 180,E1 19217.319,E2 19217.319} C_VEL
LIN {X 0,Y 586.254,Z 949.727,A -85,B 0,C 180,E1 19216.711,E2 19216.711} C_VEL
LIN {X 0,Y 583.87,Z 970.677,A -85,B 0,C 180,E1 19216.03,E2 19216.03} C_VEL
LIN {X 0,Y 581.295,Z 990.508,A -85,B 0,C 180,E1 19215.269,E2 19215.269} C_VEL
LIN {X 0,Y 578.43,Z 1010.673,A -85,B 0,C 180,E1 19214.366,E2 19214.366} C_VEL
LIN {X 0,Y 574.561,Z 1035.405,A -85,B 0,C 180,E1 19213.084,E2 19213.084} C_VEL
LIN {X 0,Y 570.611,Z 1057.78,A -85,B 0,C 180,E1 19211.713,E2 19211.713} C_VEL
LIN {X 0,Y 567.23,Z 1076.049,A -85,B 0,C 180,E1 19210.445,E2 19210.445} C_VEL
LIN {X 0,Y 563.791,Z 1093.934,A -85,B 0,C 180,E1 19209.055,E2 19209.055} C_VEL
LIN {X 0,Y 560.366,Z 1111.335,A -85,B 0,C 180,E1 19207.544,E2 19207.544} C_VEL
LIN {X 0,Y 556.636,Z 1130.172,A -85,B 0,C 180,E1 19205.715,E2 19205.715} C_VEL
LIN {X 0,Y 552.421,Z 1151.156,A -85,B 0,C 180,E1 19203.385,E2 19203.385} C_VEL
LIN {X 0,Y 549.447,Z 1166.336,A -85,B 0,C 180,E1 19201.487,E2 19201.487} C_VEL
LIN {X 0,Y 546.745,Z 1180.835,A -85,B 0,C 180,E1 19199.471,E2 19199.471} C_VEL
LIN {X 0,Y 543.874,Z 1197.221,A -85,B 0,C 180,E1 19196.918,E2 19196.918} C_VEL
LIN {X 0,Y 541.5,Z 1211.61,A -85,B 0,C 180,E1 19194.318,E2 19194.318} C_VEL
LIN {X 0,Y 539.872,Z 1222.563,A -85,B 0,C 180,E1 19192.087,E2 19192.087} C_VEL
LIN {X 0,Y 538.637,Z 1232.247,A -85,B 0,C 180,E1 19189.861,E2 19189.861} C_VEL
LIN {X 0,Y 537.452,Z 1243.082,A -85,B 0,C 180,E1 19187.008,E2 19187.008} C_VEL
LIN {X 0,Y 536.674,Z 1251.702,A -85,B 0,C 180,E1 19184.239,E2 19184.239} C_VEL
LIN {X 0,Y 536.316,Z 1257.688,A -85,B 0,C 180,E1 19181.946,E2 19181.946} C_VEL
LIN {X 0,Y 536.053,Z 1262.61,A -85,B 0,C 180,E1 19179.667,E2 19179.667} C_VEL
LIN {X 0,Y 535.961,Z 1266.454,A -85,B 0,C 180,E1 19177.399,E2 19177.399} C_VEL
LIN {X 0,Y 535.922,Z 1269.384,A -85,B 0,C 180,E1 19175.034,E2 19175.034} C_VEL
LIN {X 0,Y 535.908,Z 1271.39,A -85,B 0,C 180,E1 19172.355,E2 19172.355} C_VEL
LIN {X 0,Y 535.87,Z 1271.904,A -85,B 0,C 180,E1 19169.469,E2 19169.469} C_VEL
LIN {X 0,Y 535.909,Z 1271.113,A -85,B 0,C 180,E1 19167.116,E2 19167.116} C_VEL
LIN {X 0,Y 535.923,Z 1269.26,A -85,B 0,C 180,E1 19164.758,E2 19164.758} C_VEL
LIN {X 0,Y 535.964,Z 1266.278,A -85,B 0,C 180,E1 19162.392,E2 19162.392} C_VEL
LIN {X 0,Y 536.082,Z 1262.174,A -85,B 0,C 180,E1 19160.014,E2 19160.014} C_VEL
LIN {X 0,Y 536.431,Z 1255.871,A -85,B 0,C 180,E1 19157.188,E2 19157.188} C_VEL
LIN {X 0,Y 537.024,Z 1247.721,A -85,B 0,C 180,E1 19154.341,E2 19154.341} C_VEL
LIN {X 0,Y 537.773,Z 1239.877,A -85,B 0,C 180,E1 19152.026,E2 19152.026} C_VEL
LIN {X 0,Y 538.82,Z 1230.8,A -85,B 0,C 180,E1 19149.699,E2 19149.699} C_VEL
LIN {X 0,Y 540.348,Z 1219.387,A -85,B 0,C 180,E1 19147.137,E2 19147.137} C_VEL
LIN {X 0,Y 542.589,Z 1204.703,A -85,B 0,C 180,E1 19144.308,E2 19144.308} C_VEL
LIN {X 0,Y 544.782,Z 1191.659,A -85,B 0,C 180,E1 19142.099,E2 19142.099} C_VEL
LIN {X 0,Y 547.299,Z 1177.785,A -85,B 0,C 180,E1 19139.995,E2 19139.995} C_VEL
LIN {X 0,Y 550.771,Z 1159.919,A -85,B 0,C 180,E1 19137.584,E2 19137.584} C_VEL
LIN {X 0,Y 554.379,Z 1141.207,A -85,B 0,C 180,E1 19135.385,E2 19135.385} C_VEL
LIN {X 0,Y 557.64,Z 1124.895,A -85,B 0,C 180,E1 19133.663,E2 19133.663} C_VEL
LIN {X 0,Y 561.132,Z 1107.408,A -85,B 0,C 180,E1 19132.007,E2 19132.007} C_VEL
LIN {X 0,Y 565.63,Z 1084.632,A -85,B 0,C 180,E1 19130.104,E2 19130.104} C_VEL
LIN {X 0,Y 569.585,Z 1063.352,A -85,B 0,C 180,E1 19128.568,E2 19128.568} C_VEL
LIN {X 0,Y 572.872,Z 1044.772,A -85,B 0,C 180,E1 19127.38,E2 19127.38} C_VEL
LIN {X 0,Y 576.184,Z 1024.842,A -85,B 0,C 180,E1 19126.254,E2 19126.254} C_VEL
LIN {X 0,Y 579.694,Z 1002.114,A -85,B 0,C 180,E1 19125.14,E2 19125.14} C_VEL
LIN {X 0,Y 583.363,Z 974.944,A -85,B 0,C 180,E1 19124.033,E2 19124.033} C_VEL
LIN {X 0,Y 585.933,Z 952.635,A -85,B 0,C 180,E1 19123.285,E2 19123.285} C_VEL
LIN {X 0,Y 588.038,Z 931.502,A -85,B 0,C 180,E1 19122.705,E2 19122.705} C_VEL
LIN {X 0,Y 589.812,Z 909.579,A -85,B 0,C 180,E1 19122.223,E2 19122.223} C_VEL
LIN {X 0,Y 591.384,Z 881.37,A -85,B 0,C 180,E1 19121.754,E2 19121.754} C_VEL
LIN {X 0,Y 598.996,Z 659.061,A -85,B 0,C 180,E1 19118.544,E2 19118.544} C_VEL
LIN {X 0,Y 604.324,Z 510.744,A -85,B 0,C 180,E1 19116.352,E2 19116.352} C_VEL
LIN {X 0,Y 592.734,Z 493.595,A -85,B 0,C 180,E1 19114.44,E2 19114.44} C_VEL
LIN {X 0,Y 581.898,Z 478.392,A -85,B 0,C 180,E1 19112.507,E2 19112.507} C_VEL
LIN {X 0,Y 576.309,Z 471.122,A -85,B 0,C 180,E1 19111.453,E2 19111.453} C_VEL
LIN {X 0,Y 571.084,Z 464.68,A -85,B 0,C 180,E1 19110.427,E2 19110.427} C_VEL
LIN {X 0,Y 567.44,Z 460.16,A -85,B 0,C 180,E1 19109.68,E2 19109.68} C_VEL
LIN {X 0,Y 563.134,Z 454.861,A -85,B 0,C 180,E1 19108.763,E2 19108.763} C_VEL
LIN {X 0,Y 559.459,Z 450.479,A -85,B 0,C 180,E1 19107.95,E2 19107.95} C_VEL
LIN {X 0,Y 557.904,Z 448.741,A -85,B 0,C 180,E1 19107.6,E2 19107.6} C_VEL
LIN {X 0,Y 554.475,Z 444.631,A -85,B 0,C 180,E1 19106.797,E2 19106.797} C_VEL
LIN {X 0,Y 553.497,Z 443.332,A -85,B 0,C 180,E1 19106.558,E2 19106.558} C_VEL
LIN {X 0,Y 550.217,Z 440.144,A -85,B 0,C 180,E1 19105.771,E2 19105.771} C_VEL
LIN {X 0,Y 548.291,Z 437.159,A -85,B 0,C 180,E1 19105.261,E2 19105.261} C_VEL
LIN {X 0,Y 545.115,Z 434.598,A -85,B 0,C 180,E1 19104.462,E2 19104.462} C_VEL
LIN {X 0,Y 543.163,Z 431.048,A -85,B 0,C 180,E1 19103.891,E2 19103.891} C_VEL
LIN {X 0,Y 539.654,Z 428.747,A -85,B 0,C 180,E1 19102.956,E2 19102.956} C_VEL
LIN {X 0,Y 537.993,Z 425.993,A -85,B 0,C 180,E1 19102.439,E2 19102.439} C_VEL
LIN {X 0,Y 537.595,Z 424.247,A -85,B 0,C 180,E1 19102.241,E2 19102.241} C_VEL
LIN {X 0,Y 537.555,Z 424.231,A -85,B 0,C 180,E1 19098.884,E2 19098.884} C_VEL
LIN {X 0,Y 537.62,Z 424.208,A -85,B 0,C 180,E1 19095.645,E2 19095.645} C_VEL
LIN {X 0,Y 537.556,Z 424.259,A -85,B 0,C 180,E1 19092.461,E2 19092.461} C_VEL
LIN {X 0,Y 537.581,Z 424.203,A -85,B 0,C 180,E1 19089.097,E2 19089.097} C_VEL
LIN {X 0,Y 537.557,Z 424.27,A -85,B 0,C 180,E1 19086.086,E2 19086.086} C_VEL
LIN {X 0,Y 537.558,Z 424.205,A -85,B 0,C 180,E1 19082.665,E2 19082.665} C_VEL
LIN {X 0,Y 537.575,Z 424.271,A -85,B 0,C 180,E1 19079.574,E2 19079.574} C_VEL
LIN {X 0,Y 537.541,Z 424.21,A -85,B 0,C 180,E1 19076.16,E2 19076.16} C_VEL
LIN {X 0,Y 537.623,Z 424.247,A -85,B 0,C 180,E1 19072.842,E2 19072.842} C_VEL
LIN {X 0,Y 537.54,Z 424.219,A -85,B 0,C 180,E1 19069.605,E2 19069.605} C_VEL
LIN {X 0,Y 537.578,Z 424.227,A -85,B 0,C 180,E1 19066.336,E2 19066.336} C_VEL
LIN {X 0,Y 537.545,Z 424.234,A -85,B 0,C 180,E1 19063.243,E2 19063.243} C_VEL
LIN {X 0,Y 537.55,Z 424.21,A -85,B 0,C 180,E1 19059.872,E2 19059.872} C_VEL
LIN {X 0,Y 537.574,Z 424.315,A -85,B 0,C 180,E1 19057.931,E2 19057.931} C_VEL
LIN {X 0,Y 537.903,Z 425.804,A -85,B 0,C 180,E1 19057.7,E2 19057.7} C_VEL
LIN {X 0,Y 539.461,Z 428.548,A -85,B 0,C 180,E1 19057.208,E2 19057.208} C_VEL
LIN {X 0,Y 542.385,Z 430.612,A -85,B 0,C 180,E1 19056.419,E2 19056.419} C_VEL
LIN {X 0,Y 544.204,Z 433.35,A -85,B 0,C 180,E1 19055.899,E2 19055.899} C_VEL
LIN {X 0,Y 546.881,Z 436.312,A -85,B 0,C 180,E1 19055.19,E2 19055.19} C_VEL
LIN {X 0,Y 548.409,Z 437.803,A -85,B 0,C 180,E1 19054.803,E2 19054.803} C_VEL
LIN {X 0,Y 553.885,Z 444.654,A -85,B 0,C 180,E1 19053.433,E2 19053.433} C_VEL
LIN {X 0,Y 557.209,Z 448.517,A -85,B 0,C 180,E1 19052.653,E2 19052.653} C_VEL
LIN {X 0,Y 561.335,Z 453.568,A -85,B 0,C 180,E1 19051.717,E2 19051.717} C_VEL
LIN {X 0,Y 573.478,Z 469.447,A -85,B 0,C 180,E1 19049.162,E2 19049.162} C_VEL
LIN {X 0,Y 586.503,Z 487.372,A -85,B 0,C 180,E1 19046.704,E2 19046.704} C_VEL
LIN {X 0,Y 600.451,Z 507.862,A -85,B 0,C 180,E1 19044.32,E2 19044.32} C_VEL
LIN {X 0,Y 604.445,Z 514.401,A -85,B 0,C 180,E1 19043.669,E2 19043.669} C_VEL
LIN {X 0,Y 596.59,Z 732.843,A -85,B 0,C 180,E1 19040.47,E2 19040.47} C_VEL
LIN {X 0,Y 590.674,Z 903.219,A -85,B 0,C 180,E1 19038.003,E2 19038.003} C_VEL
LIN {X 0,Y 589.037,Z 927.687,A -85,B 0,C 180,E1 19037.553,E2 19037.553} C_VEL
LIN {X 0,Y 586.409,Z 956.096,A -85,B 0,C 180,E1 19036.839,E2 19036.839} C_VEL
LIN {X 0,Y 583.878,Z 978.429,A -85,B 0,C 180,E1 19036.127,E2 19036.127} C_VEL
LIN {X 0,Y 581.21,Z 999.138,A -85,B 0,C 180,E1 19035.339,E2 19035.339} C_VEL
LIN {X 0,Y 578.325,Z 1019.504,A -85,B 0,C 180,E1 19034.434,E2 19034.434} C_VEL
LIN {X 0,Y 574.467,Z 1044.362,A -85,B 0,C 180,E1 19033.153,E2 19033.153} C_VEL
LIN {X 0,Y 570.468,Z 1067.27,A -85,B 0,C 180,E1 19031.756,E2 19031.756} C_VEL
LIN {X 0,Y 567.026,Z 1086.083,A -85,B 0,C 180,E1 19030.455,E2 19030.455} C_VEL
LIN {X 0,Y 563.679,Z 1103.721,A -85,B 0,C 180,E1 19029.089,E2 19029.089} C_VEL
LIN {X 0,Y 560.222,Z 1121.551,A -85,B 0,C 180,E1 19027.548,E2 19027.548} C_VEL
LIN {X 0,Y 556.23,Z 1142.141,A -85,B 0,C 180,E1 19025.553,E2 19025.553} C_VEL
LIN {X 0,Y 552.342,Z 1161.544,A -85,B 0,C 180,E1 19023.384,E2 19023.384} C_VEL
LIN {X 0,Y 549.376,Z 1176.696,A -85,B 0,C 180,E1 19021.485,E2 19021.485} C_VEL
LIN {X 0,Y 546.817,Z 1190.397,A -85,B 0,C 180,E1 19019.58,E2 19019.58} C_VEL
LIN {X 0,Y 544.26,Z 1204.896,A -85,B 0,C 180,E1 19017.336,E2 19017.336} C_VEL
LIN {X 0,Y 541.629,Z 1220.713,A -85,B 0,C 180,E1 19014.538,E2 19014.538} C_VEL
LIN {X 0,Y 539.904,Z 1232.328,A -85,B 0,C 180,E1 19012.181,E2 19012.181} C_VEL
LIN {X 0,Y 538.669,Z 1241.994,A -85,B 0,C 180,E1 19009.967,E2 19009.967} C_VEL
LIN {X 0,Y 537.533,Z 1252.145,A -85,B 0,C 180,E1 19007.311,E2 19007.311} C_VEL
LIN {X 0,Y 536.713,Z 1261.239,A -85,B 0,C 180,E1 19004.452,E2 19004.452} C_VEL
LIN {X 0,Y 536.322,Z 1267.553,A -85,B 0,C 180,E1 19002.049,E2 19002.049} C_VEL
LIN {X 0,Y 536.061,Z 1272.501,A -85,B 0,C 180,E1 18999.769,E2 18999.769} C_VEL
LIN {X 0,Y 535.962,Z 1276.371,A -85,B 0,C 180,E1 18997.5,E2 18997.5} C_VEL
LIN {X 0,Y 535.924,Z 1279.326,A -85,B 0,C 180,E1 18995.135,E2 18995.135} C_VEL
LIN {X 0,Y 535.907,Z 1281.288,A -85,B 0,C 180,E1 18992.563,E2 18992.563} C_VEL
LIN {X 0,Y 535.878,Z 1281.938,A -85,B 0,C 180,E1 18989.676,E2 18989.676} C_VEL
LIN {X 0,Y 535.91,Z 1281.08,A -85,B 0,C 180,E1 18987.11,E2 18987.11} C_VEL
LIN {X 0,Y 535.924,Z 1279.204,A -85,B 0,C 180,E1 18984.752,E2 18984.752} C_VEL
LIN {X 0,Y 535.961,Z 1276.361,A -85,B 0,C 180,E1 18982.493,E2 18982.493} C_VEL
LIN {X 0,Y 536.062,Z 1272.489,A -85,B 0,C 180,E1 18980.225,E2 18980.225} C_VEL
LIN {X 0,Y 536.335,Z 1267.284,A -85,B 0,C 180,E1 18977.836,E2 18977.836} C_VEL
LIN {X 0,Y 536.881,Z 1259.673,A -85,B 0,C 180,E1 18974.994,E2 18974.994} C_VEL
LIN {X 0,Y 537.719,Z 1250.308,A -85,B 0,C 180,E1 18972.189,E2 18972.189} C_VEL
LIN {X 0,Y 538.787,Z 1241.054,A -85,B 0,C 180,E1 18969.805,E2 18969.805} C_VEL
LIN {X 0,Y 540.143,Z 1230.707,A -85,B 0,C 180,E1 18967.466,E2 18967.466} C_VEL
LIN {X 0,Y 542.402,Z 1215.884,A -85,B 0,C 180,E1 18964.561,E2 18964.561} C_VEL
LIN {X 0,Y 544.716,Z 1202.055,A -85,B 0,C 180,E1 18962.207,E2 18962.207} C_VEL
LIN {X 0,Y 547.103,Z 1188.811,A -85,B 0,C 180,E1 18960.189,E2 18960.189} C_VEL
LIN {X 0,Y 550.082,Z 1173.267,A -85,B 0,C 180,E1 18958.063,E2 18958.063} C_VEL
LIN {X 0,Y 554.074,Z 1152.806,A -85,B 0,C 180,E1 18955.607,E2 18955.607} C_VEL
LIN {X 0,Y 557.377,Z 1135.944,A -85,B 0,C 180,E1 18953.827,E2 18953.827} C_VEL
LIN {X 0,Y 560.692,Z 1119.032,A -85,B 0,C 180,E1 18952.223,E2 18952.223} C_VEL
LIN {X 0,Y 564.332,Z 1100.283,A -85,B 0,C 180,E1 18950.63,E2 18950.63} C_VEL
LIN {X 0,Y 569.021,Z 1075.226,A -85,B 0,C 180,E1 18948.772,E2 18948.772} C_VEL
LIN {X 0,Y 572.592,Z 1054.938,A -85,B 0,C 180,E1 18947.47,E2 18947.47} C_VEL
LIN {X 0,Y 575.857,Z 1035.2,A -85,B 0,C 180,E1 18946.353,E2 18946.353} C_VEL
LIN {X 0,Y 579.004,Z 1014.783,A -85,B 0,C 180,E1 18945.342,E2 18945.342} C_VEL
LIN {X 0,Y 582.494,Z 989.981,A -85,B 0,C 180,E1 18944.289,E2 18944.289} C_VEL
LIN {X 0,Y 585.611,Z 963.392,A -85,B 0,C 180,E1 18943.377,E2 18943.377} C_VEL
LIN {X 0,Y 587.798,Z 941.763,A -85,B 0,C 180,E1 18942.778,E2 18942.778} C_VEL
LIN {X 0,Y 589.563,Z 920.39,A -85,B 0,C 180,E1 18942.301,E2 18942.301} C_VEL
LIN {X 0,Y 590.965,Z 897.319,A -85,B 0,C 180,E1 18941.904,E2 18941.904} C_VEL
LIN {X 0,Y 598.571,Z 675.803,A -85,B 0,C 180,E1 18938.702,E2 18938.702} C_VEL
LIN {X 0,Y 604.375,Z 514.072,A -85,B 0,C 180,E1 18936.319,E2 18936.319} C_VEL
LIN {X 0,Y 592.417,Z 496.016,A -85,B 0,C 180,E1 18934.344,E2 18934.344} C_VEL
LIN {X 0,Y 583.114,Z 482.786,A -85,B 0,C 180,E1 18932.694,E2 18932.694} C_VEL
LIN {X 0,Y 575.223,Z 471.962,A -85,B 0,C 180,E1 18931.199,E2 18931.199} C_VEL
LIN {X 0,Y 568.083,Z 462.519,A -85,B 0,C 180,E1 18929.759,E2 18929.759} C_VEL
LIN {X 0,Y 563.986,Z 457.205,A -85,B 0,C 180,E1 18928.889,E2 18928.889} C_VEL
LIN {X 0,Y 560.516,Z 452.762,A -85,B 0,C 180,E1 18928.125,E2 18928.125} C_VEL
LIN {X 0,Y 555.819,Z 446.838,A -85,B 0,C 180,E1 18927.045,E2 18927.045} C_VEL
LIN {X 0,Y 547.375,Z 436.644,A -85,B 0,C 180,E1 18924.959,E2 18924.959} C_VEL
LIN {X 0,Y 544.466,Z 433.718,A -85,B 0,C 180,E1 18924.204,E2 18924.204} C_VEL
LIN {X 0,Y 542.664,Z 430.715,A -85,B 0,C 180,E1 18923.683,E2 18923.683} C_VEL
LIN {X 0,Y 539.531,Z 428.614,A -85,B 0,C 180,E1 18922.846,E2 18922.846} C_VEL
LIN {X 0,Y 537.924,Z 425.77,A -85,B 0,C 180,E1 18922.341,E2 18922.341} C_VEL
LIN {X 0,Y 537.61,Z 424.239,A -85,B 0,C 180,E1 18922.099,E2 18922.099} C_VEL
LIN {X 0,Y 537.562,Z 424.235,A -85,B 0,C 180,E1 18918.771,E2 18918.771} C_VEL
LIN {X 0,Y 537.615,Z 424.206,A -85,B 0,C 180,E1 18915.535,E2 18915.535} C_VEL
LIN {X 0,Y 537.588,Z 424.265,A -85,B 0,C 180,E1 18912.242,E2 18912.242} C_VEL
LIN {X 0,Y 537.575,Z 424.205,A -85,B 0,C 180,E1 18908.773,E2 18908.773} C_VEL
LIN {X 0,Y 537.628,Z 424.256,A -85,B 0,C 180,E1 18905.55,E2 18905.55} C_VEL
LIN {X 0,Y 537.586,Z 424.209,A -85,B 0,C 180,E1 18902.132,E2 18902.132} C_VEL
LIN {X 0,Y 537.603,Z 424.232,A -85,B 0,C 180,E1 18898.721,E2 18898.721} C_VEL
LIN {X 0,Y 537.618,Z 424.224,A -85,B 0,C 180,E1 18895.306,E2 18895.306} C_VEL
LIN {X 0,Y 537.596,Z 424.214,A -85,B 0,C 180,E1 18891.981,E2 18891.981} C_VEL
LIN {X 0,Y 537.618,Z 424.253,A -85,B 0,C 180,E1 18888.521,E2 18888.521} C_VEL
LIN {X 0,Y 537.61,Z 424.203,A -85,B 0,C 180,E1 18885.128,E2 18885.128} C_VEL
LIN {X 0,Y 537.61,Z 424.256,A -85,B 0,C 180,E1 18881.792,E2 18881.792} C_VEL
LIN {X 0,Y 537.619,Z 424.218,A -85,B 0,C 180,E1 18878.392,E2 18878.392} C_VEL
LIN {X 0,Y 537.638,Z 424.411,A -85,B 0,C 180,E1 18877.58,E2 18877.58} C_VEL
LIN {X 0,Y 538.628,Z 427.258,A -85,B 0,C 180,E1 18877.229,E2 18877.229} C_VEL
LIN {X 0,Y 540.884,Z 429.765,A -85,B 0,C 180,E1 18876.581,E2 18876.581} C_VEL
LIN {X 0,Y 543.229,Z 431.178,A -85,B 0,C 180,E1 18875.968,E2 18875.968} C_VEL
LIN {X 0,Y 545.292,Z 434.75,A -85,B 0,C 180,E1 18875.373,E2 18875.373} C_VEL
LIN {X 0,Y 548.763,Z 437.681,A -85,B 0,C 180,E1 18874.503,E2 18874.503} C_VEL
LIN {X 0,Y 551.379,Z 441.516,A -85,B 0,C 180,E1 18873.825,E2 18873.825} C_VEL
LIN {X 0,Y 554.203,Z 444.147,A -85,B 0,C 180,E1 18873.16,E2 18873.16} C_VEL
LIN {X 0,Y 557.29,Z 448.205,A -85,B 0,C 180,E1 18872.425,E2 18872.425} C_VEL
LIN {X 0,Y 559.386,Z 450.317,A -85,B 0,C 180,E1 18871.959,E2 18871.959} C_VEL
LIN {X 0,Y 562.949,Z 454.673,A -85,B 0,C 180,E1 18871.169,E2 18871.169} C_VEL
LIN {X 0,Y 564.769,Z 456.863,A -85,B 0,C 180,E1 18870.778,E2 18870.778} C_VEL
LIN {X 0,Y 569.578,Z 462.756,A -85,B 0,C 180,E1 18869.775,E2 18869.775} C_VEL
LIN {X 0,Y 574.754,Z 469.233,A -85,B 0,C 180,E1 18868.744,E2 18868.744} C_VEL
LIN {X 0,Y 580.679,Z 476.69,A -85,B 0,C 180,E1 18867.621,E2 18867.621} C_VEL
LIN {X 0,Y 591.711,Z 492.142,A -85,B 0,C 180,E1 18865.639,E2 18865.639} C_VEL
LIN {X 0,Y 602.759,Z 508.36,A -85,B 0,C 180,E1 18863.804,E2 18863.804} C_VEL
LIN {X 0,Y 604.376,Z 511.154,A -85,B 0,C 180,E1 18863.539,E2 18863.539} C_VEL
LIN {X 0,Y 596.631,Z 725.991,A -85,B 0,C 180,E1 18860.392,E2 18860.392} C_VEL
LIN {X 0,Y 590.749,Z 894.594,A -85,B 0,C 180,E1 18857.949,E2 18857.949} C_VEL
LIN {X 0,Y 590.599,Z 897.624,A -85,B 0,C 180,E1 18857.901,E2 18857.901} C_VEL
LIN {X 0,Y 588.977,Z 907.46,A -85,B 0,C 180,E1 18857.843,E2 18857.843} C_VEL
LIN {X 0,Y 583.897,Z 924.612,A -85,B 0,C 180,E1 18857.892,E2 18857.892} C_VEL
LIN {X 0,Y 582.548,Z 932.154,A -85,B 0,C 180,E1 18857.772,E2 18857.772} C_VEL
LIN {X 0,Y 580.352,Z 953.382,A -85,B 0,C 180,E1 18857.184,E2 18857.184} C_VEL
LIN {X 0,Y 577.564,Z 976.611,A -85,B 0,C 180,E1 18856.397,E2 18856.397} C_VEL
LIN {X 0,Y 573.836,Z 1002.887,A -85,B 0,C 180,E1 18855.312,E2 18855.312} C_VEL
LIN {X 0,Y 570.25,Z 1025.255,A -85,B 0,C 180,E1 18854.206,E2 18854.206} C_VEL
LIN {X 0,Y 566.86,Z 1044.851,A -85,B 0,C 180,E1 18853.092,E2 18853.092} C_VEL
LIN {X 0,Y 563.343,Z 1063.882,A -85,B 0,C 180,E1 18851.866,E2 18851.866} C_VEL
LIN {X 0,Y 558.98,Z 1086.38,A -85,B 0,C 180,E1 18850.223,E2 18850.223} C_VEL
LIN {X 0,Y 554.523,Z 1107.801,A -85,B 0,C 180,E1 18848.404,E2 18848.404} C_VEL
LIN {X 0,Y 550.871,Z 1125.254,A -85,B 0,C 180,E1 18846.734,E2 18846.734} C_VEL
LIN {X 0,Y 547.455,Z 1141.533,A -85,B 0,C 180,E1 18844.996,E2 18844.996} C_VEL
LIN {X 0,Y 543.596,Z 1160.412,A -85,B 0,C 180,E1 18842.739,E2 18842.739} C_VEL
LIN {X 0,Y 540.049,Z 1177.757,A -85,B 0,C 180,E1 18840.363,E2 18840.363} C_VEL
LIN {X 0,Y 537.466,Z 1191.092,A -85,B 0,C 180,E1 18838.322,E2 18838.322} C_VEL
LIN {X 0,Y 535.222,Z 1203.737,A -85,B 0,C 180,E1 18836.163,E2 18836.163} C_VEL
LIN {X 0,Y 532.913,Z 1217.932,A -85,B 0,C 180,E1 18833.436,E2 18833.436} C_VEL
LIN {X 0,Y 531.087,Z 1230.415,A -85,B 0,C 180,E1 18830.616,E2 18830.616} C_VEL
LIN {X 0,Y 529.949,Z 1239.529,A -85,B 0,C 180,E1 18828.255,E2 18828.255} C_VEL
LIN {X 0,Y 529.106,Z 1247.766,A -85,B 0,C 180,E1 18825.793,E2 18825.793} C_VEL
LIN {X 0,Y 528.448,Z 1256.159,A -85,B 0,C 180,E1 18822.793,E2 18822.793} C_VEL
LIN {X 0,Y 528.107,Z 1262.195,A -85,B 0,C 180,E1 18820.034,E2 18820.034} C_VEL
LIN {X 0,Y 527.959,Z 1266.292,A -85,B 0,C 180,E1 18817.621,E2 18817.621} C_VEL
LIN {X 0,Y 527.925,Z 1269.268,A -85,B 0,C 180,E1 18815.219,E2 18815.219} C_VEL
LIN {X 0,Y 527.909,Z 1271.188,A -85,B 0,C 180,E1 18812.717,E2 18812.717} C_VEL
LIN {X 0,Y 527.889,Z 1271.971,A -85,B 0,C 180,E1 18809.786,E2 18809.786} C_VEL
LIN {X 0,Y 527.91,Z 1271.113,A -85,B 0,C 180,E1 18807.072,E2 18807.072} C_VEL
LIN {X 0,Y 527.924,Z 1269.256,A -85,B 0,C 180,E1 18804.678,E2 18804.678} C_VEL
LIN {X 0,Y 527.963,Z 1266.274,A -85,B 0,C 180,E1 18802.276,E2 18802.276} C_VEL
LIN {X 0,Y 528.109,Z 1262.169,A -85,B 0,C 180,E1 18799.862,E2 18799.862} C_VEL
LIN {X 0,Y 528.48,Z 1255.87,A -85,B 0,C 180,E1 18796.992,E2 18796.992} C_VEL
LIN {X 0,Y 529.104,Z 1247.718,A -85,B 0,C 180,E1 18794.101,E2 18794.101} C_VEL
LIN {X 0,Y 529.917,Z 1239.873,A -85,B 0,C 180,E1 18791.751,E2 18791.751} C_VEL
LIN {X 0,Y 531.056,Z 1230.653,A -85,B 0,C 180,E1 18789.354,E2 18789.354} C_VEL
LIN {X 0,Y 532.755,Z 1218.862,A -85,B 0,C 180,E1 18786.676,E2 18786.676} C_VEL
LIN {X 0,Y 535.133,Z 1204.249,A -85,B 0,C 180,E1 18783.839,E2 18783.839} C_VEL
LIN {X 0,Y 537.393,Z 1191.488,A -85,B 0,C 180,E1 18781.652,E2 18781.652} C_VEL
LIN {X 0,Y 540.083,Z 1177.595,A -85,B 0,C 180,E1 18779.523,E2 18779.523} C_VEL
LIN {X 0,Y 543.806,Z 1159.288,A -85,B 0,C 180,E1 18777.032,E2 18777.032} C_VEL
LIN {X 0,Y 547.505,Z 1141.292,A -85,B 0,C 180,E1 18774.887,E2 18774.887} C_VEL
LIN {X 0,Y 550.875,Z 1125.237,A -85,B 0,C 180,E1 18773.174,E2 18773.174} C_VEL
LIN {X 0,Y 554.463,Z 1108.097,A -85,B 0,C 180,E1 18771.532,E2 18771.532} C_VEL
LIN {X 0,Y 559.06,Z 1086.005,A -85,B 0,C 180,E1 18769.657,E2 18769.657} C_VEL
LIN {X 0,Y 563.336,Z 1063.945,A -85,B 0,C 180,E1 18768.048,E2 18768.048} C_VEL
LIN {X 0,Y 566.859,Z 1044.85,A -85,B 0,C 180,E1 18766.818,E2 18766.818} C_VEL
LIN {X 0,Y 570.258,Z 1025.192,A -85,B 0,C 180,E1 18765.701,E2 18765.701} C_VEL
LIN {X 0,Y 573.801,Z 1003.105,A -85,B 0,C 180,E1 18764.609,E2 18764.609} C_VEL
LIN {X 0,Y 577.671,Z 975.756,A -85,B 0,C 180,E1 18763.482,E2 18763.482} C_VEL
LIN {X 0,Y 580.393,Z 953.032,A -85,B 0,C 180,E1 18762.715,E2 18762.715} C_VEL
LIN {X 0,Y 582.57,Z 931.961,A -85,B 0,C 180,E1 18762.133,E2 18762.133} C_VEL
LIN {X 0,Y 584.394,Z 910.292,A -85,B 0,C 180,E1 18761.653,E2 18761.653} C_VEL
LIN {X 0,Y 586.009,Z 883.143,A -85,B 0,C 180,E1 18761.194,E2 18761.194} C_VEL
LIN {X 0,Y 593.943,Z 661.279,A -85,B 0,C 180,E1 18757.97,E2 18757.97} C_VEL
LIN {X 0,Y 599.427,Z 514.903,A -85,B 0,C 180,E1 18755.794,E2 18755.794} C_VEL
LIN {X 0,Y 588.803,Z 499.13,A -85,B 0,C 180,E1 18753.995,E2 18753.995} C_VEL
LIN {X 0,Y 578.464,Z 484.486,A -85,B 0,C 180,E1 18752.109,E2 18752.109} C_VEL
LIN {X 0,Y 573.167,Z 477.609,A -85,B 0,C 180,E1 18751.089,E2 18751.089} C_VEL
LIN {X 0,Y 565.175,Z 467.53,A -85,B 0,C 180,E1 18749.461,E2 18749.461} C_VEL
LIN {X 0,Y 560.257,Z 461.617,A -85,B 0,C 180,E1 18748.4,E2 18748.4} C_VEL
LIN {X 0,Y 555.72,Z 456.105,A -85,B 0,C 180,E1 18747.369,E2 18747.369} C_VEL
LIN {X 0,Y 552.024,Z 451.667,A -85,B 0,C 180,E1 18746.49,E2 18746.49} C_VEL
LIN {X 0,Y 550.536,Z 450.116,A -85,B 0,C 180,E1 18746.132,E2 18746.132} C_VEL
LIN {X 0,Y 547.273,Z 446.333,A -85,B 0,C 180,E1 18745.311,E2 18745.311} C_VEL
LIN {X 0,Y 545.99,Z 444.52,A -85,B 0,C 180,E1 18744.969,E2 18744.969} C_VEL
LIN {X 0,Y 542.7,Z 441.51,A -85,B 0,C 180,E1 18744.115,E2 18744.115} C_VEL
LIN {X 0,Y 540.739,Z 438.331,A -85,B 0,C 180,E1 18743.541,E2 18743.541} C_VEL
LIN {X 0,Y 537.489,Z 435.918,A -85,B 0,C 180,E1 18742.649,E2 18742.649} C_VEL
LIN {X 0,Y 535.51,Z 432.487,A -85,B 0,C 180,E1 18742.014,E2 18742.014} C_VEL
LIN {X 0,Y 535.298,Z 431.884,A -85,B 0,C 180,E1 18741.937,E2 18741.937} C_VEL
LIN {X 0,Y 532.045,Z 430.019,A -85,B 0,C 180,E1 18740.978,E2 18740.978} C_VEL
LIN {X 0,Y 530.234,Z 427.396,A -85,B 0,C 180,E1 18740.36,E2 18740.36} C_VEL
LIN {X 0,Y 529.659,Z 425.193,A -85,B 0,C 180,E1 18740.095,E2 18740.095} C_VEL
LIN {X 0,Y 529.616,Z 425.237,A -85,B 0,C 180,E1 18736.79,E2 18736.79} C_VEL
LIN {X 0,Y 529.677,Z 425.201,A -85,B 0,C 180,E1 18733.537,E2 18733.537} C_VEL
LIN {X 0,Y 529.611,Z 425.214,A -85,B 0,C 180,E1 18730.332,E2 18730.332} C_VEL
LIN {X 0,Y 529.636,Z 425.227,A -85,B 0,C 180,E1 18726.94,E2 18726.94} C_VEL
LIN {X 0,Y 529.624,Z 425.2,A -85,B 0,C 180,E1 18723.789,E2 18723.789} C_VEL
LIN {X 0,Y 529.612,Z 425.251,A -85,B 0,C 180,E1 18720.325,E2 18720.325} C_VEL
LIN {X 0,Y 529.665,Z 425.188,A -85,B 0,C 180,E1 18717.078,E2 18717.078} C_VEL
LIN {X 0,Y 529.608,Z 425.261,A -85,B 0,C 180,E1 18713.822,E2 18713.822} C_VEL
LIN {X 0,Y 529.645,Z 425.189,A -85,B 0,C 180,E1 18710.547,E2 18710.547} C_VEL
LIN {X 0,Y 529.613,Z 425.254,A -85,B 0,C 180,E1 18707.349,E2 18707.349} C_VEL
LIN {X 0,Y 529.605,Z 425.204,A -85,B 0,C 180,E1 18703.887,E2 18703.887} C_VEL
LIN {X 0,Y 529.632,Z 425.212,A -85,B 0,C 180,E1 18700.823,E2 18700.823} C_VEL
LIN {X 0,Y 529.637,Z 425.305,A -85,B 0,C 180,E1 18700.005,E2 18700.005} C_VEL
LIN {X 0,Y 530.493,Z 428.002,A -85,B 0,C 180,E1 18699.65,E2 18699.65} C_VEL
LIN {X 0,Y 532.681,Z 430.559,A -85,B 0,C 180,E1 18698.933,E2 18698.933} C_VEL
LIN {X 0,Y 535.352,Z 432.116,A -85,B 0,C 180,E1 18698.15,E2 18698.15} C_VEL
LIN {X 0,Y 537.216,Z 435.602,A -85,B 0,C 180,E1 18697.541,E2 18697.541} C_VEL
LIN {X 0,Y 540.339,Z 438.154,A -85,B 0,C 180,E1 18696.671,E2 18696.671} C_VEL
LIN {X 0,Y 541.224,Z 439.146,A -85,B 0,C 180,E1 18696.423,E2 18696.423} C_VEL
LIN {X 0,Y 543.857,Z 442.873,A -85,B 0,C 180,E1 18695.68,E2 18695.68} C_VEL
LIN {X 0,Y 546.312,Z 445.203,A -85,B 0,C 180,E1 18695.047,E2 18695.047} C_VEL
LIN {X 0,Y 554.918,Z 455.856,A -85,B 0,C 180,E1 18692.908,E2 18692.908} C_VEL
LIN {X 0,Y 560.336,Z 462.806,A -85,B 0,C 180,E1 18691.662,E2 18691.662} C_VEL
LIN {X 0,Y 568.271,Z 473.1,A -85,B 0,C 180,E1 18689.961,E2 18689.961} C_VEL
LIN {X 0,Y 578.427,Z 487.043,A -85,B 0,C 180,E1 18687.948,E2 18687.948} C_VEL
LIN {X 0,Y 588.035,Z 500.8,A -85,B 0,C 180,E1 18686.189,E2 18686.189} C_VEL
LIN {X 0,Y 599.556,Z 518.307,A -85,B 0,C 180,E1 18684.23,E2 18684.23} C_VEL
LIN {X 0,Y 591.412,Z 735.315,A -85,B 0,C 180,E1 18681.034,E2 18681.034} C_VEL
LIN {X 0,Y 585.33,Z 903.092,A -85,B 0,C 180,E1 18678.589,E2 18678.589} C_VEL
LIN {X 0,Y 583.631,Z 927.609,A -85,B 0,C 180,E1 18678.137,E2 18678.137} C_VEL
LIN {X 0,Y 580.906,Z 956.013,A -85,B 0,C 180,E1 18677.421,E2 18677.421} C_VEL
LIN {X 0,Y 578.279,Z 978.344,A -85,B 0,C 180,E1 18676.707,E2 18676.707} C_VEL
LIN {X 0,Y 575.512,Z 999.051,A -85,B 0,C 180,E1 18675.916,E2 18675.916} C_VEL
LIN {X 0,Y 572.508,Z 1019.352,A -85,B 0,C 180,E1 18675.012,E2 18675.012} C_VEL
LIN {X 0,Y 568.48,Z 1044.272,A -85,B 0,C 180,E1 18673.722,E2 18673.722} C_VEL
LIN {X 0,Y 564.317,Z 1067.18,A -85,B 0,C 180,E1 18672.316,E2 18672.316} C_VEL
LIN {X 0,Y 560.721,Z 1085.992,A -85,B 0,C 180,E1 18671.006,E2 18671.006} C_VEL
LIN {X 0,Y 557.221,Z 1103.629,A -85,B 0,C 180,E1 18669.631,E2 18669.631} C_VEL
LIN {X 0,Y 553.477,Z 1122.07,A -85,B 0,C 180,E1 18668.021,E2 18668.021} C_VEL
LIN {X 0,Y 549.175,Z 1143.199,A -85,B 0,C 180,E1 18665.939,E2 18665.939} C_VEL
LIN {X 0,Y 545.281,Z 1161.81,A -85,B 0,C 180,E1 18663.832,E2 18663.832} C_VEL
LIN {X 0,Y 542.299,Z 1176.39,A -85,B 0,C 180,E1 18661.989,E2 18661.989} C_VEL
LIN {X 0,Y 539.517,Z 1190.395,A -85,B 0,C 180,E1 18660.021,E2 18660.021} C_VEL
LIN {X 0,Y 536.848,Z 1204.667,A -85,B 0,C 180,E1 18657.785,E2 18657.785} C_VEL
LIN {X 0,Y 534.017,Z 1220.711,A -85,B 0,C 180,E1 18654.911,E2 18654.911} C_VEL
LIN {X 0,Y 532.201,Z 1232.273,A -85,B 0,C 180,E1 18652.532,E2 18652.532} C_VEL
LIN {X 0,Y 530.815,Z 1242.451,A -85,B 0,C 180,E1 18650.16,E2 18650.16} C_VEL
LIN {X 0,Y 529.581,Z 1252.953,A -85,B 0,C 180,E1 18647.352,E2 18647.352} C_VEL
LIN {X 0,Y 528.757,Z 1261.542,A -85,B 0,C 180,E1 18644.563,E2 18644.563} C_VEL
LIN {X 0,Y 528.339,Z 1267.807,A -85,B 0,C 180,E1 18642.123,E2 18642.123} C_VEL
LIN {X 0,Y 528.069,Z 1272.705,A -85,B 0,C 180,E1 18639.808,E2 18639.808} C_VEL
LIN {X 0,Y 527.964,Z 1276.528,A -85,B 0,C 180,E1 18637.505,E2 18637.505} C_VEL
LIN {X 0,Y 527.924,Z 1279.436,A -85,B 0,C 180,E1 18635.104,E2 18635.104} C_VEL
LIN {X 0,Y 527.909,Z 1281.55,A -85,B 0,C 180,E1 18632.168,E2 18632.168} C_VEL
LIN {X 0,Y 527.865,Z 1281.871,A -85,B 0,C 180,E1 18629.346,E2 18629.346} C_VEL
LIN {X 0,Y 527.91,Z 1281.08,A -85,B 0,C 180,E1 18627.066,E2 18627.066} C_VEL
LIN {X 0,Y 527.925,Z 1279.201,A -85,B 0,C 180,E1 18624.672,E2 18624.672} C_VEL
LIN {X 0,Y 527.96,Z 1276.358,A -85,B 0,C 180,E1 18622.379,E2 18622.379} C_VEL
LIN {X 0,Y 528.085,Z 1272.486,A -85,B 0,C 180,E1 18620.076,E2 18620.076} C_VEL
LIN {X 0,Y 528.367,Z 1267.284,A -85,B 0,C 180,E1 18617.65,E2 18617.65} C_VEL
LIN {X 0,Y 528.964,Z 1259.673,A -85,B 0,C 180,E1 18614.764,E2 18614.764} C_VEL
LIN {X 0,Y 529.844,Z 1250.499,A -85,B 0,C 180,E1 18611.969,E2 18611.969} C_VEL
LIN {X 0,Y 530.939,Z 1241.511,A -85,B 0,C 180,E1 18609.608,E2 18609.608} C_VEL
LIN {X 0,Y 532.368,Z 1231.22,A -85,B 0,C 180,E1 18607.236,E2 18607.236} C_VEL
LIN {X 0,Y 534.541,Z 1217.786,A -85,B 0,C 180,E1 18604.516,E2 18604.516} C_VEL
LIN {X 0,Y 537.166,Z 1202.753,A -85,B 0,C 180,E1 18601.903,E2 18601.903} C_VEL
LIN {X 0,Y 539.676,Z 1189.58,A -85,B 0,C 180,E1 18599.859,E2 18599.859} C_VEL
LIN {X 0,Y 542.61,Z 1174.955,A -85,B 0,C 180,E1 18597.82,E2 18597.82} C_VEL
LIN {X 0,Y 546.368,Z 1156.783,A -85,B 0,C 180,E1 18595.562,E2 18595.562} C_VEL
LIN {X 0,Y 550.415,Z 1136.857,A -85,B 0,C 180,E1 18593.412,E2 18593.412} C_VEL
LIN {X 0,Y 553.972,Z 1119.552,A -85,B 0,C 180,E1 18591.748,E2 18591.748} C_VEL
LIN {X 0,Y 557.77,Z 1100.862,A -85,B 0,C 180,E1 18590.141,E2 18590.141} C_VEL
LIN {X 0,Y 562.359,Z 1077.659,A -85,B 0,C 180,E1 18588.386,E2 18588.386} C_VEL
LIN {X 0,Y 566.385,Z 1055.743,A -85,B 0,C 180,E1 18586.96,E2 18586.96} C_VEL
LIN {X 0,Y 569.773,Z 1036.118,A -85,B 0,C 180,E1 18585.836,E2 18585.836} C_VEL
LIN {X 0,Y 573.014,Z 1015.965,A -85,B 0,C 180,E1 18584.827,E2 18584.827} C_VEL
LIN {X 0,Y 576.088,Z 995.038,A -85,B 0,C 180,E1 18583.92,E2 18583.92} C_VEL
LIN {X 0,Y 579.532,Z 968.568,A -85,B 0,C 180,E1 18582.958,E2 18582.958} C_VEL
LIN {X 0,Y 582.189,Z 943.39,A -85,B 0,C 180,E1 18582.238,E2 18582.238} C_VEL
LIN {X 0,Y 584.073,Z 921.637,A -85,B 0,C 180,E1 18581.744,E2 18581.744} C_VEL
LIN {X 0,Y 585.509,Z 899.486,A -85,B 0,C 180,E1 18581.354,E2 18581.354} C_VEL
LIN {X 0,Y 593.373,Z 681.088,A -85,B 0,C 180,E1 18578.174,E2 18578.174} C_VEL
LIN {X 0,Y 599.489,Z 518.226,A -85,B 0,C 180,E1 18575.765,E2 18575.765} C_VEL
LIN {X 0,Y 586.676,Z 498.773,A -85,B 0,C 180,E1 18573.577,E2 18573.577} C_VEL
LIN {X 0,Y 576.417,Z 484.273,A -85,B 0,C 180,E1 18571.68,E2 18571.68} C_VEL
LIN {X 0,Y 566.462,Z 470.736,A -85,B 0,C 180,E1 18569.678,E2 18569.678} C_VEL
LIN {X 0,Y 558.199,Z 460.017,A -85,B 0,C 180,E1 18567.874,E2 18567.874} C_VEL
LIN {X 0,Y 553.243,Z 453.79,A -85,B 0,C 180,E1 18566.716,E2 18566.716} C_VEL
LIN {X 0,Y 545.283,Z 444.063,A -85,B 0,C 180,E1 18564.714,E2 18564.714} C_VEL
LIN {X 0,Y 542.232,Z 440.864,A -85,B 0,C 180,E1 18563.905,E2 18563.905} C_VEL
LIN {X 0,Y 540.609,Z 438.279,A -85,B 0,C 180,E1 18563.432,E2 18563.432} C_VEL
LIN {X 0,Y 537.449,Z 435.875,A -85,B 0,C 180,E1 18562.564,E2 18562.564} C_VEL
LIN {X 0,Y 535.542,Z 432.574,A -85,B 0,C 180,E1 18561.955,E2 18561.955} C_VEL
LIN {X 0,Y 535.157,Z 431.838,A -85,B 0,C 180,E1 18561.828,E2 18561.828} C_VEL
LIN {X 0,Y 531.908,Z 429.882,A -85,B 0,C 180,E1 18560.869,E2 18560.869} C_VEL
LIN {X 0,Y 530.182,Z 427.241,A -85,B 0,C 180,E1 18560.276,E2 18560.276} C_VEL
LIN {X 0,Y 529.67,Z 425.193,A -85,B 0,C 180,E1 18560.037,E2 18560.037} C_VEL
LIN {X 0,Y 529.626,Z 425.233,A -85,B 0,C 180,E1 18556.789,E2 18556.789} C_VEL
LIN {X 0,Y 529.672,Z 425.208,A -85,B 0,C 180,E1 18553.426,E2 18553.426} C_VEL
LIN {X 0,Y 529.644,Z 425.204,A -85,B 0,C 180,E1 18550.222,E2 18550.222} C_VEL
LIN {X 0,Y 529.647,Z 425.242,A -85,B 0,C 180,E1 18546.722,E2 18546.722} C_VEL
LIN {X 0,Y 529.678,Z 425.185,A -85,B 0,C 180,E1 18543.355,E2 18543.355} C_VEL
LIN {X 0,Y 529.661,Z 425.256,A -85,B 0,C 180,E1 18540,E2 18540} C_VEL
LIN {X 0,Y 529.655,Z 425.188,A -85,B 0,C 180,E1 18536.537,E2 18536.537} C_VEL
LIN {X 0,Y 529.683,Z 425.238,A -85,B 0,C 180,E1 18533.17,E2 18533.17} C_VEL
LIN {X 0,Y 529.664,Z 425.199,A -85,B 0,C 180,E1 18529.779,E2 18529.779} C_VEL
LIN {X 0,Y 529.673,Z 425.206,A -85,B 0,C 180,E1 18526.351,E2 18526.351} C_VEL
LIN {X 0,Y 529.674,Z 425.231,A -85,B 0,C 180,E1 18522.986,E2 18522.986} C_VEL
LIN {X 0,Y 529.694,Z 425.383,A -85,B 0,C 180,E1 18519.739,E2 18519.739} C_VEL
LIN {X 0,Y 530.618,Z 428.081,A -85,B 0,C 180,E1 18519.367,E2 18519.367} C_VEL
LIN {X 0,Y 532.99,Z 430.746,A -85,B 0,C 180,E1 18518.6,E2 18518.6} C_VEL
LIN {X 0,Y 535.417,Z 432.112,A -85,B 0,C 180,E1 18517.895,E2 18517.895} C_VEL
LIN {X 0,Y 537.297,Z 435.615,A -85,B 0,C 180,E1 18517.285,E2 18517.285} C_VEL
LIN {X 0,Y 540.339,Z 438.124,A -85,B 0,C 180,E1 18516.44,E2 18516.44} C_VEL
LIN {X 0,Y 541.154,Z 438.875,A -85,B 0,C 180,E1 18516.218,E2 18516.218} C_VEL
LIN {X 0,Y 543.688,Z 442.621,A -85,B 0,C 180,E1 18515.499,E2 18515.499} C_VEL
LIN {X 0,Y 546.553,Z 445.103,A -85,B 0,C 180,E1 18514.769,E2 18514.769} C_VEL
LIN {X 0,Y 549.548,Z 449.179,A -85,B 0,C 180,E1 18513.992,E2 18513.992} C_VEL
LIN {X 0,Y 551.938,Z 451.522,A -85,B 0,C 180,E1 18513.419,E2 18513.419} C_VEL
LIN {X 0,Y 555.526,Z 455.955,A -85,B 0,C 180,E1 18512.563,E2 18512.563} C_VEL
LIN {X 0,Y 557.271,Z 457.971,A -85,B 0,C 180,E1 18512.163,E2 18512.163} C_VEL
LIN {X 0,Y 562.408,Z 464.191,A -85,B 0,C 180,E1 18511.022,E2 18511.022} C_VEL
LIN {X 0,Y 567.283,Z 470.234,A -85,B 0,C 180,E1 18509.991,E2 18509.991} C_VEL
LIN {X 0,Y 575.317,Z 480.242,A -85,B 0,C 180,E1 18508.393,E2 18508.393} C_VEL
LIN {X 0,Y 584.543,Z 492.981,A -85,B 0,C 180,E1 18506.666,E2 18506.666} C_VEL
LIN {X 0,Y 596.189,Z 509.933,A -85,B 0,C 180,E1 18504.647,E2 18504.647} C_VEL
LIN {X 0,Y 599.482,Z 515.336,A -85,B 0,C 180,E1 18504.095,E2 18504.095} C_VEL
LIN {X 0,Y 591.42,Z 729.669,A -85,B 0,C 180,E1 18500.939,E2 18500.939} C_VEL
LIN {X 0,Y 585.408,Z 894.712,A -85,B 0,C 180,E1 18498.532,E2 18498.532} C_VEL
LIN {X 0,Y 583.728,Z 919.198,A -85,B 0,C 180,E1 18498.077,E2 18498.077} C_VEL
LIN {X 0,Y 582.548,Z 932.154,A -85,B 0,C 180,E1 18497.772,E2 18497.772} C_VEL
LIN {X 0,Y 581.079,Z 939.7,A -85,B 0,C 180,E1 18497.668,E2 18497.668} C_VEL
LIN {X 0,Y 574.712,Z 959.924,A -85,B 0,C 180,E1 18497.52,E2 18497.52} C_VEL
LIN {X 0,Y 573.377,Z 966.175,A -85,B 0,C 180,E1 18497.362,E2 18497.362} C_VEL
LIN {X 0,Y 570.369,Z 988.149,A -85,B 0,C 180,E1 18496.534,E2 18496.534} C_VEL
LIN {X 0,Y 567.226,Z 1008.623,A -85,B 0,C 180,E1 18495.628,E2 18495.628} C_VEL
LIN {X 0,Y 563.676,Z 1029.633,A -85,B 0,C 180,E1 18494.554,E2 18494.554} C_VEL
LIN {X 0,Y 559.161,Z 1054.286,A -85,B 0,C 180,E1 18493.087,E2 18493.087} C_VEL
LIN {X 0,Y 554.739,Z 1076.249,A -85,B 0,C 180,E1 18491.554,E2 18491.554} C_VEL
LIN {X 0,Y 550.921,Z 1094.468,A -85,B 0,C 180,E1 18490.115,E2 18490.115} C_VEL
LIN {X 0,Y 547.064,Z 1112.37,A -85,B 0,C 180,E1 18488.531,E2 18488.531} C_VEL
LIN {X 0,Y 542.602,Z 1133.059,A -85,B 0,C 180,E1 18486.464,E2 18486.464} C_VEL
LIN {X 0,Y 538.308,Z 1152.236,A -85,B 0,C 180,E1 18484.251,E2 18484.251} C_VEL
LIN {X 0,Y 535.037,Z 1167.246,A -85,B 0,C 180,E1 18482.311,E2 18482.311} C_VEL
LIN {X 0,Y 531.863,Z 1182.381,A -85,B 0,C 180,E1 18480.131,E2 18480.131} C_VEL
LIN {X 0,Y 528.422,Z 1199.93,A -85,B 0,C 180,E1 18477.255,E2 18477.255} C_VEL
LIN {X 0,Y 526.081,Z 1212.76,A -85,B 0,C 180,E1 18474.839,E2 18474.839} C_VEL
LIN {X 0,Y 524.373,Z 1223.136,A -85,B 0,C 180,E1 18472.644,E2 18472.644} C_VEL
LIN {X 0,Y 522.863,Z 1233.682,A -85,B 0,C 180,E1 18470.122,E2 18470.122} C_VEL
LIN {X 0,Y 521.484,Z 1244.943,A -85,B 0,C 180,E1 18466.947,E2 18466.947} C_VEL
LIN {X 0,Y 520.786,Z 1252.008,A -85,B 0,C 180,E1 18464.57,E2 18464.57} C_VEL
LIN {X 0,Y 520.374,Z 1257.691,A -85,B 0,C 180,E1 18462.318,E2 18462.318} C_VEL
LIN {X 0,Y 520.099,Z 1262.607,A -85,B 0,C 180,E1 18459.966,E2 18459.966} C_VEL
LIN {X 0,Y 519.961,Z 1266.45,A -85,B 0,C 180,E1 18457.628,E2 18457.628} C_VEL
LIN {X 0,Y 519.925,Z 1269.38,A -85,B 0,C 180,E1 18455.189,E2 18455.189} C_VEL
LIN {X 0,Y 519.908,Z 1271.391,A -85,B 0,C 180,E1 18452.428,E2 18452.428} C_VEL
LIN {X 0,Y 519.869,Z 1271.904,A -85,B 0,C 180,E1 18449.452,E2 18449.452} C_VEL
LIN {X 0,Y 519.91,Z 1271.112,A -85,B 0,C 180,E1 18447.027,E2 18447.027} C_VEL
LIN {X 0,Y 519.926,Z 1269.252,A -85,B 0,C 180,E1 18444.596,E2 18444.596} C_VEL
LIN {X 0,Y 519.966,Z 1266.43,A -85,B 0,C 180,E1 18442.268,E2 18442.268} C_VEL
LIN {X 0,Y 520.119,Z 1262.372,A -85,B 0,C 180,E1 18439.817,E2 18439.817} C_VEL
LIN {X 0,Y 520.46,Z 1256.637,A -85,B 0,C 180,E1 18437.127,E2 18437.127} C_VEL
LIN {X 0,Y 521.156,Z 1248.15,A -85,B 0,C 180,E1 18433.992,E2 18433.992} C_VEL
LIN {X 0,Y 522.064,Z 1239.822,A -85,B 0,C 180,E1 18431.453,E2 18431.453} C_VEL
LIN {X 0,Y 523.26,Z 1230.791,A -85,B 0,C 180,E1 18429.068,E2 18429.068} C_VEL
LIN {X 0,Y 525.005,Z 1219.377,A -85,B 0,C 180,E1 18426.429,E2 18426.429} C_VEL
LIN {X 0,Y 527.504,Z 1204.878,A -85,B 0,C 180,E1 18423.553,E2 18423.553} C_VEL
LIN {X 0,Y 529.872,Z 1192.202,A -85,B 0,C 180,E1 18421.34,E2 18421.34} C_VEL
LIN {X 0,Y 532.529,Z 1179.13,A -85,B 0,C 180,E1 18419.294,E2 18419.294} C_VEL
LIN {X 0,Y 535.858,Z 1163.617,A -85,B 0,C 180,E1 18417.107,E2 18417.107} C_VEL
LIN {X 0,Y 540.25,Z 1143.394,A -85,B 0,C 180,E1 18414.605,E2 18414.605} C_VEL
LIN {X 0,Y 544.027,Z 1126.17,A -85,B 0,C 180,E1 18412.734,E2 18412.734} C_VEL
LIN {X 0,Y 547.704,Z 1109.392,A -85,B 0,C 180,E1 18411.103,E2 18411.103} C_VEL
LIN {X 0,Y 551.868,Z 1090.112,A -85,B 0,C 180,E1 18409.431,E2 18409.431} C_VEL
LIN {X 0,Y 556.861,Z 1065.939,A -85,B 0,C 180,E1 18407.611,E2 18407.611} C_VEL
LIN {X 0,Y 560.735,Z 1045.827,A -85,B 0,C 180,E1 18406.299,E2 18406.299} C_VEL
LIN {X 0,Y 564.308,Z 1025.999,A -85,B 0,C 180,E1 18405.16,E2 18405.16} C_VEL
LIN {X 0,Y 567.889,Z 1004.523,A -85,B 0,C 180,E1 18404.087,E2 18404.087} C_VEL
LIN {X 0,Y 571.827,Z 978.195,A -85,B 0,C 180,E1 18402.978,E2 18402.978} C_VEL
LIN {X 0,Y 574.863,Z 953.861,A -85,B 0,C 180,E1 18402.147,E2 18402.147} C_VEL
LIN {X 0,Y 577.149,Z 932.553,A -85,B 0,C 180,E1 18401.553,E2 18401.553} C_VEL
